      $ 538 "Direction: Base Z+"
      global move_thread_flag_538=0
      thread move_thread_538():
        enter_critical
        move_thread_flag_538 = 1
        local towardsPos=calculate_point_to_move_towards(p[0.0,0.0,0.0,0.0,0.0,0.0], [0.0,0.0,1.0], 0.06)
        movel(towardsPos, a=0.035, v=0.03)
        move_thread_flag_538 = 2
        exit_critical
      end
      move_thread_flag_538 = 0
      move_thread_han_538 = run move_thread_538()
      while (True):
        sleep(1.0E-10)
        if (move_thread_flag_538 > 1):
          join move_thread_han_538
          $ 539 "Until (distance)"
          break
        end
        sync()
      end
      $ 540 "Set CO[1]=Apagar"
      set_configurable_digital_out(1, False)
      $ 541 "barreno_actual≔barreno_actual+1"
      global barreno_actual=barreno_actual+1
      $ 542 "Call Quitar_broca"
      Quitar_broca()
      $ 543 "Call Poner_broca"
      Poner_broca()
    end
    $ 544 "CD"
    $ 545 "'desbaste_inicial'"
    # 'desbaste_inicial'
    $ 546 "bajada_broca≔p[0,0,-0.012,0,0,0]"
    global bajada_broca=p[0,0,-0.012,0,0,0]
    $ 547 "barrenos_menos1≔8"
    global barrenos_menos1=8
    $ 548 "barreno_actual≔0"
    global barreno_actual=0
    $ 549 "Loop barreno_actual≤barrenos_menos1"
    while (barreno_actual <= barrenos_menos1):
      $ 550 "Perforacion"
      $ 551 "MoveL"
      $ 552 "internos≔interpolate_pose(Linea1_C, Linea1_D, barreno_actual/barrenos_menos1)"
      global internos= interpolate_pose (Linea1_C_p, Linea1_D_p, barreno_actual/barrenos_menos1)
      $ 553 "internos" "breakAfter"
      movel(internos, a=0.5, v=0.1)
      $ 554 "'desbaste_inicial'"
      # 'desbaste_inicial'
      $ 555 "bajada_broca≔p[0,0,-0.024,0,0,0]"
      global bajada_broca=p[0,0,-0.024,0,0,0]
      $ 556 "bajada≔p[0,0,0.024,0,0,0]"
      global bajada=p[0,0,0.024,0,0,0]
      $ 557 "Direction: Base Z-"
      global move_thread_flag_557=0
      thread move_thread_557():
        enter_critical
        move_thread_flag_557 = 1
        local towardsPos=calculate_point_to_move_towards(p[0.0,0.0,0.0,0.0,0.0,0.0], [0.0,0.0,-1.0], 0.072)
        movel(towardsPos, a=0.035, v=0.03)
        move_thread_flag_557 = 2
        exit_critical
      end
      move_thread_flag_557 = 0
      move_thread_han_557 = run move_thread_557()
      while (True):
        sleep(1.0E-10)
        if (move_thread_flag_557 > 1):
          join move_thread_han_557
          $ 558 "Until (distance)"
          break
        end
        sync()
      end
      $ 559 "Popup: punto contacto alanzdo"
      popup("punto contacto alanzdo", "Mensaje", False, False, blocking=True)
      $ 560 "Direction: Base Z+"
      global move_thread_flag_560=0
      thread move_thread_560():
        enter_critical
        move_thread_flag_560 = 1
        local towardsPos=calculate_point_to_move_towards(p[0.0,0.0,0.0,0.0,0.0,0.0], [0.0,0.0,1.0], 0.002)
        movel(towardsPos, a=0.005, v=0.003)
        move_thread_flag_560 = 2
        exit_critical
      end
      move_thread_flag_560 = 0
      move_thread_han_560 = run move_thread_560()
      while (True):
        sleep(1.0E-10)
        if (move_thread_flag_560 > 1):
          join move_thread_han_560
          $ 561 "Until (distance)"
          break
        end
        sync()
      end
      $ 562 "Wait: 0.3"
      sleep(0.3)
      $ 563 "Set CO[1]=Encender"
      set_configurable_digital_out(1, True)
      $ 564 "Wait: 0.3"
      sleep(0.3)
      $ 565 "Loop 1 times"
      Loop_85 = 0
      while (Loop_85 < 1):
        $ 566 "bajar≔pose_add(get_actual_tcp_pose(), bajada_broca)"
        global bajar= pose_add ( get_actual_tcp_pose (), bajada_broca)
        $ 567 "bajar" "breakAfter"
        movel(bajar, a=0.005, v=0.001)
        $ 568 "subir≔pose_sub(get_actual_tcp_pose(), bajada_broca)"
        global subir= pose_sub ( get_actual_tcp_pose (), bajada_broca)
        $ 569 "subir" "breakAfter"
        movel(subir, a=0.01, v=0.005)
        $ 570 "bajada_broca≔pose_sub(bajada_broca, bajada)"
        global bajada_broca= pose_sub (bajada_broca, bajada)
        Loop_85 = Loop_85 + 1
      end
      $ 571 "Direction: Base Z+"
      global move_thread_flag_571=0
      thread move_thread_571():
        enter_critical
        move_thread_flag_571 = 1
        local towardsPos=calculate_point_to_move_towards(p[0.0,0.0,0.0,0.0,0.0,0.0], [0.0,0.0,1.0], 0.06)
        movel(towardsPos, a=0.035, v=0.03)
        move_thread_flag_571 = 2
        exit_critical
      end
      move_thread_flag_571 = 0
      move_thread_han_571 = run move_thread_571()
      while (True):
        sleep(1.0E-10)
        if (move_thread_flag_571 > 1):
          join move_thread_han_571
          $ 572 "Until (distance)"
          break
        end
        sync()
      end
      $ 573 "Set CO[1]=Apagar"
      set_configurable_digital_out(1, False)
      $ 574 "barreno_actual≔barreno_actual+1"
      global barreno_actual=barreno_actual+1
      $ 575 "Call Quitar_broca"
      Quitar_broca()
      $ 576 "Call Poner_broca"
      Poner_broca()
    end
    $ 577 "EF"
    $ 578 "'desbaste_inicial'"
    # 'desbaste_inicial'
    $ 579 "bajada_broca≔p[0,0,-0.012,0,0,0]"
    global bajada_broca=p[0,0,-0.012,0,0,0]
    $ 580 "barrenos_menos1≔8"
    global barrenos_menos1=8
    $ 581 "barreno_actual≔0"
    global barreno_actual=0
    $ 582 "Loop barreno_actual≤barrenos_menos1"
    while (barreno_actual <= barrenos_menos1):
      $ 583 "Perforacion"
      $ 584 "MoveL"
      $ 585 "internos≔interpolate_pose(Linea1_E, Linea1_F, barreno_actual/barrenos_menos1)"
      global internos= interpolate_pose (Linea1_E_p, Linea1_F_p, barreno_actual/barrenos_menos1)
      $ 586 "internos" "breakAfter"
      movel(internos, a=0.5, v=0.1)
      $ 587 "'desbaste_inicial'"
      # 'desbaste_inicial'
      $ 588 "bajada_broca≔p[0,0,-0.024,0,0,0]"
      global bajada_broca=p[0,0,-0.024,0,0,0]
      $ 589 "bajada≔p[0,0,0.024,0,0,0]"
      global bajada=p[0,0,0.024,0,0,0]
      $ 590 "Direction: Base Z-"
      global move_thread_flag_590=0
      thread move_thread_590():
        enter_critical
        move_thread_flag_590 = 1
        local towardsPos=calculate_point_to_move_towards(p[0.0,0.0,0.0,0.0,0.0,0.0], [0.0,0.0,-1.0], 0.072)
        movel(towardsPos, a=0.035, v=0.03)
        move_thread_flag_590 = 2
        exit_critical
      end
      move_thread_flag_590 = 0
      move_thread_han_590 = run move_thread_590()
      while (True):
        sleep(1.0E-10)
        if (move_thread_flag_590 > 1):
          join move_thread_han_590
          $ 591 "Until (distance)"
          break
        end
        sync()
      end
      $ 592 "Popup: punto contacto alanzdo"
      popup("punto contacto alanzdo", "Mensaje", False, False, blocking=True)
      $ 593 "Direction: Base Z+"
      global move_thread_flag_593=0
      thread move_thread_593():
        enter_critical
        move_thread_flag_593 = 1
        local towardsPos=calculate_point_to_move_towards(p[0.0,0.0,0.0,0.0,0.0,0.0], [0.0,0.0,1.0], 0.002)
        movel(towardsPos, a=0.005, v=0.003)
        move_thread_flag_593 = 2
        exit_critical
      end
      move_thread_flag_593 = 0
      move_thread_han_593 = run move_thread_593()
      while (True):
        sleep(1.0E-10)
        if (move_thread_flag_593 > 1):
          join move_thread_han_593
          $ 594 "Until (distance)"
          break
        end
        sync()
      end
      $ 595 "Wait: 0.3"
      sleep(0.3)
      $ 596 "Set CO[1]=Encender"
      set_configurable_digital_out(1, True)
      $ 597 "Wait: 0.3"
      sleep(0.3)
      $ 598 "Loop 1 times"
      Loop_87 = 0
      while (Loop_87 < 1):
        $ 599 "bajar≔pose_add(get_actual_tcp_pose(), bajada_broca)"
        global bajar= pose_add ( get_actual_tcp_pose (), bajada_broca)
        $ 600 "bajar" "breakAfter"
        movel(bajar, a=0.005, v=0.001)
        $ 601 "subir≔pose_sub(get_actual_tcp_pose(), bajada_broca)"
        global subir= pose_sub ( get_actual_tcp_pose (), bajada_broca)
        $ 602 "subir" "breakAfter"
        movel(subir, a=0.01, v=0.005)
        $ 603 "bajada_broca≔pose_sub(bajada_broca, bajada)"
        global bajada_broca= pose_sub (bajada_broca, bajada)
        Loop_87 = Loop_87 + 1
      end
      $ 604 "Direction: Base Z+"
      global move_thread_flag_604=0
      thread move_thread_604():
        enter_critical
        move_thread_flag_604 = 1
        local towardsPos=calculate_point_to_move_towards(p[0.0,0.0,0.0,0.0,0.0,0.0], [0.0,0.0,1.0], 0.06)
        movel(towardsPos, a=0.035, v=0.03)
        move_thread_flag_604 = 2
        exit_critical
      end
      move_thread_flag_604 = 0
      move_thread_han_604 = run move_thread_604()
      while (True):
        sleep(1.0E-10)
        if (move_thread_flag_604 > 1):
          join move_thread_han_604
          $ 605 "Until (distance)"
          break
        end
        sync()
      end
      $ 606 "Set CO[1]=Apagar"
      set_configurable_digital_out(1, False)
      $ 607 "barreno_actual≔barreno_actual+1"
      global barreno_actual=barreno_actual+1
      $ 608 "Call Quitar_broca"
      Quitar_broca()
      $ 609 "Call Poner_broca"
      Poner_broca()
    end
    $ 610 "Popup: Linea1 con full Terminada!"
    popup("Linea1 con full Terminada!", "Mensaje", False, False, blocking=True)
    $ 611 "Linea2"
    $ 612 "Marcar_puntos"
    $ 613 "MoveL"
    $ 614 "Home2" "breakAfter"
    movel(Home2_p, a=0.5, v=0.1)
    $ 623 "Linea2_A" "breakAfter"
    movel(Linea2_A_p, a=0.5, v=0.1)
    $ 624 "Linea2_B" "breakAfter"
    movel(Linea2_B_p, a=0.5, v=0.1)
    $ 625 "Linea2_C" "breakAfter"
    movel(Linea2_C_p, a=0.5, v=0.1)
    $ 626 "Linea2_D" "breakAfter"
    movel(Linea2_D_p, a=0.5, v=0.1)
    $ 627 "Linea2_E" "breakAfter"
    movel(Linea2_E_p, a=0.5, v=0.1)
    $ 628 "Linea2_F" "breakAfter"
    movel(Linea2_F_p, a=0.5, v=0.1)
    $ 629 "AB"
    $ 630 "'desbaste_inicial'"
    # 'desbaste_inicial'
    $ 631 "bajada_broca≔p[0,0,-0.012,0,0,0]"
    global bajada_broca=p[0,0,-0.012,0,0,0]
    $ 632 "barrenos_menos1≔8"
    global barrenos_menos1=8
    $ 633 "barreno_actual≔1"
    global barreno_actual=1
    $ 634 "Loop barreno_actual≤barrenos_menos1"
    while (barreno_actual <= barrenos_menos1):
      $ 635 "Perforacion"
      $ 636 "MoveL"
      $ 637 "internos≔interpolate_pose(Linea2_A, Linea2_B, barreno_actual/barrenos_menos1)"
      global internos= interpolate_pose (Linea2_A_p, Linea2_B_p, barreno_actual/barrenos_menos1)
      $ 638 "internos" "breakAfter"
      movel(internos, a=0.5, v=0.1)
      $ 639 "'desbaste_inicial'"
      # 'desbaste_inicial'
      $ 640 "bajada_broca≔p[0,0,-0.024,0,0,0]"
      global bajada_broca=p[0,0,-0.024,0,0,0]
      $ 641 "bajada≔p[0,0,0.024,0,0,0]"
      global bajada=p[0,0,0.024,0,0,0]
      $ 642 "Direction: Base Z-"
      global move_thread_flag_642=0
      thread move_thread_642():
        enter_critical
        move_thread_flag_642 = 1
        local towardsPos=calculate_point_to_move_towards(p[0.0,0.0,0.0,0.0,0.0,0.0], [0.0,0.0,-1.0], 0.076)
        movel(towardsPos, a=0.035, v=0.03)
        move_thread_flag_642 = 2
        exit_critical
      end
      move_thread_flag_642 = 0
      move_thread_han_642 = run move_thread_642()
      while (True):
        sleep(1.0E-10)
        if (move_thread_flag_642 > 1):
          join move_thread_han_642
          $ 643 "Until (distance)"
          break
        end
        sync()
      end
      $ 644 "Popup: punto contacto alanzdo"
      popup("punto contacto alanzdo", "Mensaje", False, False, blocking=True)
      $ 645 "Direction: Base Z+"
      global move_thread_flag_645=0
      thread move_thread_645():
        enter_critical
        move_thread_flag_645 = 1
        local towardsPos=calculate_point_to_move_towards(p[0.0,0.0,0.0,0.0,0.0,0.0], [0.0,0.0,1.0], 0.002)
        movel(towardsPos, a=0.005, v=0.003)
        move_thread_flag_645 = 2
        exit_critical
      end
      move_thread_flag_645 = 0
      move_thread_han_645 = run move_thread_645()
      while (True):
        sleep(1.0E-10)
        if (move_thread_flag_645 > 1):
          join move_thread_han_645
          $ 646 "Until (distance)"
          break
        end
        sync()
      end
      $ 647 "Wait: 0.3"
      sleep(0.3)
      $ 648 "Set CO[1]=Encender"
      set_configurable_digital_out(1, True)
      $ 649 "Wait: 0.3"
      sleep(0.3)
      $ 650 "Loop 1 times"
      Loop_90 = 0
      while (Loop_90 < 1):
        $ 651 "bajar≔pose_add(get_actual_tcp_pose(), bajada_broca)"
        global bajar= pose_add ( get_actual_tcp_pose (), bajada_broca)
        $ 652 "bajar" "breakAfter"
        movel(bajar, a=0.005, v=0.001)
        $ 653 "subir≔pose_sub(get_actual_tcp_pose(), bajada_broca)"
        global subir= pose_sub ( get_actual_tcp_pose (), bajada_broca)
        $ 654 "subir" "breakAfter"
        movel(subir, a=0.01, v=0.005)
        $ 655 "bajada_broca≔pose_sub(bajada_broca, bajada)"
        global bajada_broca= pose_sub (bajada_broca, bajada)
        Loop_90 = Loop_90 + 1
      end
      $ 656 "Direction: Base Z+"
      global move_thread_flag_656=0
      thread move_thread_656():
        enter_critical
        move_thread_flag_656 = 1
        local towardsPos=calculate_point_to_move_towards(p[0.0,0.0,0.0,0.0,0.0,0.0], [0.0,0.0,1.0], 0.06)
        movel(towardsPos, a=0.035, v=0.03)
        move_thread_flag_656 = 2
        exit_critical
      end
      move_thread_flag_656 = 0
      move_thread_han_656 = run move_thread_656()
      while (True):
        sleep(1.0E-10)
        if (move_thread_flag_656 > 1):
          join move_thread_han_656
          $ 657 "Until (distance)"
          break
        end
        sync()
      end
      $ 658 "Set CO[1]=Apagar"
      set_configurable_digital_out(1, False)
      $ 659 "barreno_actual≔barreno_actual+1"
      global barreno_actual=barreno_actual+1
      $ 660 "Call Quitar_broca"
      Quitar_broca()
      $ 661 "Call Poner_broca"
      Poner_broca()
    end
    $ 662 "CD"
    $ 663 "'desbaste_inicial'"
    # 'desbaste_inicial'
    $ 664 "bajada_broca≔p[0,0,-0.012,0,0,0]"
    global bajada_broca=p[0,0,-0.012,0,0,0]
    $ 665 "barrenos_menos1≔8"
    global barrenos_menos1=8
    $ 666 "barreno_actual≔0"
    global barreno_actual=0
    $ 667 "Loop barreno_actual≤barrenos_menos1"
    while (barreno_actual <= barrenos_menos1):
      $ 668 "Perforacion"
      $ 669 "MoveL"
      $ 670 "internos≔interpolate_pose(Linea2_C, Linea2_D, barreno_actual/barrenos_menos1)"
      global internos= interpolate_pose (Linea2_C_p, Linea2_D_p, barreno_actual/barrenos_menos1)
      $ 671 "internos" "breakAfter"
      movel(internos, a=0.5, v=0.1)
      $ 672 "'desbaste_inicial'"
      # 'desbaste_inicial'
      $ 673 "bajada_broca≔p[0,0,-0.024,0,0,0]"
      global bajada_broca=p[0,0,-0.024,0,0,0]
      $ 674 "bajada≔p[0,0,0.024,0,0,0]"
      global bajada=p[0,0,0.024,0,0,0]
      $ 675 "Direction: Base Z-"
      global move_thread_flag_675=0
      thread move_thread_675():
        enter_critical
        move_thread_flag_675 = 1
        local towardsPos=calculate_point_to_move_towards(p[0.0,0.0,0.0,0.0,0.0,0.0], [0.0,0.0,-1.0], 0.076)
        movel(towardsPos, a=0.035, v=0.03)
        move_thread_flag_675 = 2
        exit_critical
      end
      move_thread_flag_675 = 0
      move_thread_han_675 = run move_thread_675()
      while (True):
        sleep(1.0E-10)
        if (move_thread_flag_675 > 1):
          join move_thread_han_675
          $ 676 "Until (distance)"
          break
        end
        sync()
      end
      $ 677 "Popup: punto contacto alanzdo"
      popup("punto contacto alanzdo", "Mensaje", False, False, blocking=True)
      $ 678 "Direction: Base Z+"
      global move_thread_flag_678=0
      thread move_thread_678():
        enter_critical
        move_thread_flag_678 = 1
        local towardsPos=calculate_point_to_move_towards(p[0.0,0.0,0.0,0.0,0.0,0.0], [0.0,0.0,1.0], 0.002)
        movel(towardsPos, a=0.005, v=0.003)
        move_thread_flag_678 = 2
        exit_critical
      end
      move_thread_flag_678 = 0
      move_thread_han_678 = run move_thread_678()
      while (True):
        sleep(1.0E-10)
        if (move_thread_flag_678 > 1):
          join move_thread_han_678
          $ 679 "Until (distance)"
          break
        end
        sync()
      end
      $ 680 "Wait: 0.3"
      sleep(0.3)
      $ 681 "Set CO[1]=Encender"
      set_configurable_digital_out(1, True)
      $ 682 "Wait: 0.3"
      sleep(0.3)
      $ 683 "Loop 1 times"
      Loop_92 = 0
      while (Loop_92 < 1):
        $ 684 "bajar≔pose_add(get_actual_tcp_pose(), bajada_broca)"
        global bajar= pose_add ( get_actual_tcp_pose (), bajada_broca)
        $ 685 "bajar" "breakAfter"
        movel(bajar, a=0.005, v=0.001)
        $ 686 "subir≔pose_sub(get_actual_tcp_pose(), bajada_broca)"
        global subir= pose_sub ( get_actual_tcp_pose (), bajada_broca)
        $ 687 "subir" "breakAfter"
        movel(subir, a=0.01, v=0.005)
        $ 688 "bajada_broca≔pose_sub(bajada_broca, bajada)"
        global bajada_broca= pose_sub (bajada_broca, bajada)
        Loop_92 = Loop_92 + 1
      end
      $ 689 "Direction: Base Z+"
      global move_thread_flag_689=0
      thread move_thread_689():
        enter_critical
        move_thread_flag_689 = 1
        local towardsPos=calculate_point_to_move_towards(p[0.0,0.0,0.0,0.0,0.0,0.0], [0.0,0.0,1.0], 0.06)
        movel(towardsPos, a=0.035, v=0.03)
        move_thread_flag_689 = 2
        exit_critical
      end
      move_thread_flag_689 = 0
      move_thread_han_689 = run move_thread_689()
      while (True):
        sleep(1.0E-10)
        if (move_thread_flag_689 > 1):
          join move_thread_han_689
          $ 690 "Until (distance)"
          break
        end
        sync()
      end
      $ 691 "Set CO[1]=Apagar"
      set_configurable_digital_out(1, False)
      $ 692 "barreno_actual≔barreno_actual+1"
      global barreno_actual=barreno_actual+1
      $ 693 "Call Quitar_broca"
      Quitar_broca()
      $ 694 "Call Poner_broca"
      Poner_broca()
    end
    $ 695 "EF"
    $ 696 "'desbaste_inicial'"
    # 'desbaste_inicial'
    $ 697 "bajada_broca≔p[0,0,-0.012,0,0,0]"
    global bajada_broca=p[0,0,-0.012,0,0,0]
    $ 698 "barrenos_menos1≔8"
    global barrenos_menos1=8
    $ 699 "barreno_actual≔0"
    global barreno_actual=0
    $ 700 "Loop barreno_actual≤barrenos_menos1"
    while (barreno_actual <= barrenos_menos1):
      $ 701 "Perforacion"
      $ 702 "MoveL"
      $ 703 "internos≔interpolate_pose(Linea2_E, Linea2_F, barreno_actual/barrenos_menos1)"
      global internos= interpolate_pose (Linea2_E_p, Linea2_F_p, barreno_actual/barrenos_menos1)
      $ 704 "internos" "breakAfter"
      movel(internos, a=0.5, v=0.1)
      $ 705 "'desbaste_inicial'"
      # 'desbaste_inicial'
      $ 706 "bajada_broca≔p[0,0,-0.024,0,0,0]"
      global bajada_broca=p[0,0,-0.024,0,0,0]
      $ 707 "bajada≔p[0,0,0.024,0,0,0]"
      global bajada=p[0,0,0.024,0,0,0]
      $ 708 "Direction: Base Z-"
      global move_thread_flag_708=0
      thread move_thread_708():
        enter_critical
        move_thread_flag_708 = 1
        local towardsPos=calculate_point_to_move_towards(p[0.0,0.0,0.0,0.0,0.0,0.0], [0.0,0.0,-1.0], 0.076)
        movel(towardsPos, a=0.035, v=0.03)
        move_thread_flag_708 = 2
        exit_critical
      end
      move_thread_flag_708 = 0
      move_thread_han_708 = run move_thread_708()
      while (True):
        sleep(1.0E-10)
        if (move_thread_flag_708 > 1):
          join move_thread_han_708
          $ 709 "Until (distance)"
          break
        end
        sync()
      end
      $ 710 "Popup: punto contacto alanzdo"
      popup("punto contacto alanzdo", "Mensaje", False, False, blocking=True)
      $ 711 "Direction: Base Z+"
      global move_thread_flag_711=0
      thread move_thread_711():
        enter_critical
        move_thread_flag_711 = 1
        local towardsPos=calculate_point_to_move_towards(p[0.0,0.0,0.0,0.0,0.0,0.0], [0.0,0.0,1.0], 0.002)
        movel(towardsPos, a=0.015, v=0.015)
        move_thread_flag_711 = 2
        exit_critical
      end
      move_thread_flag_711 = 0
      move_thread_han_711 = run move_thread_711()
      while (True):
        sleep(1.0E-10)
        if (move_thread_flag_711 > 1):
          join move_thread_han_711
          $ 712 "Until (distance)"
          break
        end
        sync()
      end
      $ 713 "Wait: 0.3"
      sleep(0.3)
      $ 714 "Set CO[1]=Encender"
      set_configurable_digital_out(1, True)
      $ 715 "Wait: 0.3"
      sleep(0.3)
      $ 716 "Loop 1 times"
      Loop_94 = 0
      while (Loop_94 < 1):
        $ 717 "bajar≔pose_add(get_actual_tcp_pose(), bajada_broca)"
        global bajar= pose_add ( get_actual_tcp_pose (), bajada_broca)
        $ 718 "bajar" "breakAfter"
        movel(bajar, a=0.005, v=0.001)
        $ 719 "subir≔pose_sub(get_actual_tcp_pose(), bajada_broca)"
        global subir= pose_sub ( get_actual_tcp_pose (), bajada_broca)
        $ 720 "subir" "breakAfter"
        movel(subir, a=0.01, v=0.005)
        $ 721 "bajada_broca≔pose_sub(bajada_broca, bajada)"
        global bajada_broca= pose_sub (bajada_broca, bajada)
        Loop_94 = Loop_94 + 1
      end
      $ 722 "Direction: Base Z+"
      global move_thread_flag_722=0
      thread move_thread_722():
        enter_critical
        move_thread_flag_722 = 1
        local towardsPos=calculate_point_to_move_towards(p[0.0,0.0,0.0,0.0,0.0,0.0], [0.0,0.0,1.0], 0.06)
        movel(towardsPos, a=0.035, v=0.03)
        move_thread_flag_722 = 2
        exit_critical
      end
      move_thread_flag_722 = 0
      move_thread_han_722 = run move_thread_722()
      while (True):
        sleep(1.0E-10)
        if (move_thread_flag_722 > 1):
          join move_thread_han_722
          $ 723 "Until (distance)"
          break
        end
        sync()
      end
      $ 724 "Set CO[1]=Apagar"
      set_configurable_digital_out(1, False)
      $ 725 "barreno_actual≔barreno_actual+1"
      global barreno_actual=barreno_actual+1
      $ 726 "If barreno_actual>barrenos_menos1"
      if (barreno_actual>barrenos_menos1):
        $ 727 "cambiar_broca≔ True "
        global cambiar_broca=  True
      end
      $ 728 "Call Quitar_broca"
      Quitar_broca()
      $ 729 "Call Poner_broca"
      Poner_broca()
    end
    $ 730 "Popup: Linea2 con full Terminada!"
    popup("Linea2 con full Terminada!", "Mensaje", False, False, blocking=True)
    $ 731 "600"
    $ 1243 "Broca_1"
    $ 1244 "Linea7"
    $ 1245 "Marcar_puntos"
    $ 1246 "MoveL"
    $ 1247 "Home2" "breakAfter"
    movel(Home2_p, a=0.5, v=0.1)
    $ 1248 "Linea7_A" "breakAfter"
    movel(Linea7_A_p, a=0.5, v=0.1)
    $ 1249 "bajada_comprobacion"
    $ 1250 "Direction: Base Z-"
    global move_thread_flag_1250=0
    thread move_thread_1250():
      enter_critical
      move_thread_flag_1250 = 1
      local towardsPos=calculate_point_to_move_towards(p[0.0,0.0,0.0,0.0,0.0,0.0], [0.0,0.0,-1.0], 0.071)
      movel(towardsPos, a=0.15, v=0.1)
      move_thread_flag_1250 = 2
      exit_critical
    end
    move_thread_flag_1250 = 0
    move_thread_han_1250 = run move_thread_1250()
    while (True):
      sleep(1.0E-10)
      if (move_thread_flag_1250 > 1):
        join move_thread_han_1250
        $ 1251 "Until (distance)"
        break
      end
      sync()
    end
    $ 1252 "Direction: Base Z-"
    global move_thread_flag_1252=0
    thread move_thread_1252():
      enter_critical
      move_thread_flag_1252 = 1
      local towardsPos=calculate_point_to_move_towards(p[0.0,0.0,0.0,0.0,0.0,0.0], [0.0,0.0,-1.0], 1000.0)
      movel(towardsPos, a=0.007, v=0.007)
      move_thread_flag_1252 = 2
      exit_critical
    end
    move_thread_flag_1252 = 0
    move_thread_han_1252 = run move_thread_1252()
    while (True):
      local targetTcpDirection=get_target_tcp_speed()
      local stepsToRetract=tool_contact(direction=targetTcpDirection)
      if (stepsToRetract > 0):
        kill move_thread_han_1252
        stopl(0.02)
        local backTrackMovement=get_actual_joint_positions_history(stepsToRetract)
        local contactPose=get_forward_kin(backTrackMovement)
        local posDir=[targetTcpDirection[0],targetTcpDirection[1],targetTcpDirection[2]]
        local retractTo=contactPose
        if (norm(posDir) > 1e-6):
          local normalizedPosDir=normalize(posDir)
          local additionalRetraction=p[normalizedPosDir[0] * 0.0, normalizedPosDir[1] * 0.0, normalizedPosDir[2] * 0.0, 0, 0, 0]
          retractTo = pose_sub(contactPose, additionalRetraction)
        end
        movel(retractTo, a=0.02, v=0.1)
        $ 1253 "Until (tool_contact_detection)"
        break
      end
      sync()
    end
    $ 1254 "Direction: Base Z+"
    global move_thread_flag_1254=0
    thread move_thread_1254():
      enter_critical
      move_thread_flag_1254 = 1
      local towardsPos=calculate_point_to_move_towards(p[0.0,0.0,0.0,0.0,0.0,0.0], [0.0,0.0,1.0], 0.08)
      movel(towardsPos, a=0.15, v=0.1)
      move_thread_flag_1254 = 2
      exit_critical
    end
    move_thread_flag_1254 = 0
    move_thread_han_1254 = run move_thread_1254()
    while (True):
      sleep(1.0E-10)
      if (move_thread_flag_1254 > 1):
        join move_thread_han_1254
        $ 1255 "Until (distance)"
        break
      end
      sync()
    end
    $ 1256 "Linea7_B" "breakAfter"
    movel(Linea7_B_p, a=0.5, v=0.1)
    $ 1257 "bajada_comprobacion"
    $ 1258 "Direction: Base Z-"
    global move_thread_flag_1258=0
    thread move_thread_1258():
      enter_critical
      move_thread_flag_1258 = 1
      local towardsPos=calculate_point_to_move_towards(p[0.0,0.0,0.0,0.0,0.0,0.0], [0.0,0.0,-1.0], 0.071)
      movel(towardsPos, a=0.15, v=0.1)
      move_thread_flag_1258 = 2
      exit_critical
    end
    move_thread_flag_1258 = 0
    move_thread_han_1258 = run move_thread_1258()
    while (True):
      sleep(1.0E-10)
      if (move_thread_flag_1258 > 1):
        join move_thread_han_1258
        $ 1259 "Until (distance)"
        break
      end
      sync()
    end
    $ 1260 "Direction: Base Z-"
    global move_thread_flag_1260=0
    thread move_thread_1260():
      enter_critical
      move_thread_flag_1260 = 1
      local towardsPos=calculate_point_to_move_towards(p[0.0,0.0,0.0,0.0,0.0,0.0], [0.0,0.0,-1.0], 1000.0)
      movel(towardsPos, a=0.007, v=0.007)
      move_thread_flag_1260 = 2
      exit_critical
    end
    move_thread_flag_1260 = 0
    move_thread_han_1260 = run move_thread_1260()
    while (True):
      local targetTcpDirection=get_target_tcp_speed()
      local stepsToRetract=tool_contact(direction=targetTcpDirection)
      if (stepsToRetract > 0):
        kill move_thread_han_1260
        stopl(0.02)
        local backTrackMovement=get_actual_joint_positions_history(stepsToRetract)
        local contactPose=get_forward_kin(backTrackMovement)
        local posDir=[targetTcpDirection[0],targetTcpDirection[1],targetTcpDirection[2]]
        local retractTo=contactPose
        if (norm(posDir) > 1e-6):
          local normalizedPosDir=normalize(posDir)
          local additionalRetraction=p[normalizedPosDir[0] * 0.0, normalizedPosDir[1] * 0.0, normalizedPosDir[2] * 0.0, 0, 0, 0]
          retractTo = pose_sub(contactPose, additionalRetraction)
        end
        movel(retractTo, a=0.02, v=0.1)
        $ 1261 "Until (tool_contact_detection)"
        break
      end
      sync()
    end
    $ 1262 "Direction: Base Z+"
    global move_thread_flag_1262=0
    thread move_thread_1262():
      enter_critical
      move_thread_flag_1262 = 1
      local towardsPos=calculate_point_to_move_towards(p[0.0,0.0,0.0,0.0,0.0,0.0], [0.0,0.0,1.0], 0.08)
      movel(towardsPos, a=0.15, v=0.1)
      move_thread_flag_1262 = 2
      exit_critical
    end
    move_thread_flag_1262 = 0
    move_thread_han_1262 = run move_thread_1262()
    while (True):
      sleep(1.0E-10)
      if (move_thread_flag_1262 > 1):
        join move_thread_han_1262
        $ 1263 "Until (distance)"
        break
      end
      sync()
    end
    $ 1264 "AB"
    $ 1265 "'desbaste_inicial'"
    # 'desbaste_inicial'
    $ 1266 "bajada_broca≔p[0,0,-0.008,0,0,0]"
    global bajada_broca=p[0,0,-0.008,0,0,0]
    $ 1267 "barrenos_menos1≔2"
    global barrenos_menos1=2
    $ 1268 "barreno_actual≔0"
    global barreno_actual=0
    $ 1269 "Loop barreno_actual≤barrenos_menos1"
    while (barreno_actual <= barrenos_menos1):
      $ 1270 "Perforacion"
      $ 1271 "MoveL"
      $ 1272 "internos≔interpolate_pose(Linea7_A, Linea7_B, barreno_actual/barrenos_menos1)"
      global internos= interpolate_pose (Linea7_A_p, Linea7_B_p, barreno_actual/barrenos_menos1)
      $ 1273 "internos" "breakAfter"
      movel(internos, a=0.5, v=0.1)
      $ 1274 "'desbaste_inicial'"
      # 'desbaste_inicial'
      $ 1275 "bajada_broca≔p[0,0,-0.024,0,0,0]"
      global bajada_broca=p[0,0,-0.024,0,0,0]
      $ 1276 "bajada≔p[0,0,0.024,0,0,0]"
      global bajada=p[0,0,0.024,0,0,0]
      $ 1277 "Direction: Base Z-"
      global move_thread_flag_1277=0
      thread move_thread_1277():
        enter_critical
        move_thread_flag_1277 = 1
        local towardsPos=calculate_point_to_move_towards(p[0.0,0.0,0.0,0.0,0.0,0.0], [0.0,0.0,-1.0], 0.071)
        movel(towardsPos, a=0.15, v=0.1)
        move_thread_flag_1277 = 2
        exit_critical
      end
      move_thread_flag_1277 = 0
      move_thread_han_1277 = run move_thread_1277()
      while (True):
        sleep(1.0E-10)
        if (move_thread_flag_1277 > 1):
          join move_thread_han_1277
          $ 1278 "Until (distance)"
          break
        end
        sync()
      end
      $ 1279 "Direction: Base Z-"
      global move_thread_flag_1279=0
      thread move_thread_1279():
        enter_critical
        move_thread_flag_1279 = 1
        local towardsPos=calculate_point_to_move_towards(p[0.0,0.0,0.0,0.0,0.0,0.0], [0.0,0.0,-1.0], 1000.0)
        movel(towardsPos, a=0.007, v=0.007)
        move_thread_flag_1279 = 2
        exit_critical
      end
      move_thread_flag_1279 = 0
      move_thread_han_1279 = run move_thread_1279()
      while (True):
        local targetTcpDirection=get_target_tcp_speed()
        local stepsToRetract=tool_contact(direction=targetTcpDirection)
        if (stepsToRetract > 0):
          kill move_thread_han_1279
          stopl(0.02)
          local backTrackMovement=get_actual_joint_positions_history(stepsToRetract)
          local contactPose=get_forward_kin(backTrackMovement)
          local posDir=[targetTcpDirection[0],targetTcpDirection[1],targetTcpDirection[2]]
          local retractTo=contactPose
          if (norm(posDir) > 1e-6):
            local normalizedPosDir=normalize(posDir)
            local additionalRetraction=p[normalizedPosDir[0] * 0.0, normalizedPosDir[1] * 0.0, normalizedPosDir[2] * 0.0, 0, 0, 0]
            retractTo = pose_sub(contactPose, additionalRetraction)
          end
          movel(retractTo, a=0.02, v=0.1)
          $ 1280 "Until (tool_contact_detection)"
          break
        end
        sync()
      end
      $ 1281 "Popup: punto contacto alanzdo"
      popup("punto contacto alanzdo", "Mensaje", False, False, blocking=True)
      $ 1282 "Direction: Base Z+"
      global move_thread_flag_1282=0
      thread move_thread_1282():
        enter_critical
        move_thread_flag_1282 = 1
        local towardsPos=calculate_point_to_move_towards(p[0.0,0.0,0.0,0.0,0.0,0.0], [0.0,0.0,1.0], 0.002)
        movel(towardsPos, a=0.005, v=0.003)
        move_thread_flag_1282 = 2
        exit_critical
      end
      move_thread_flag_1282 = 0
      move_thread_han_1282 = run move_thread_1282()
      while (True):
        sleep(1.0E-10)
        if (move_thread_flag_1282 > 1):
          join move_thread_han_1282
          $ 1283 "Until (distance)"
          break
        end
        sync()
      end
      $ 1284 "Wait: 0.3"
      sleep(0.3)
      $ 1285 "Set CO[1]=Encender"
      set_configurable_digital_out(1, True)
      $ 1286 "Wait: 0.3"
      sleep(0.3)
      $ 1287 "Loop 1 times"
      Loop_96 = 0
      while (Loop_96 < 1):
        $ 1288 "bajar≔pose_add(get_actual_tcp_pose(), bajada_broca)"
        global bajar= pose_add ( get_actual_tcp_pose (), bajada_broca)
        $ 1289 "bajar" "breakAfter"
        movel(bajar, a=0.01, v=0.01)
        $ 1290 "subir≔pose_sub(get_actual_tcp_pose(), bajada_broca)"
        global subir= pose_sub ( get_actual_tcp_pose (), bajada_broca)
        $ 1291 "subir" "breakAfter"
        movel(subir, a=0.015, v=0.015)
        $ 1292 "bajada_broca≔pose_sub(bajada_broca, bajada)"
        global bajada_broca= pose_sub (bajada_broca, bajada)
        Loop_96 = Loop_96 + 1
      end
      $ 1293 "Direction: Base Z+"
      global move_thread_flag_1293=0
      thread move_thread_1293():
        enter_critical
        move_thread_flag_1293 = 1
        local towardsPos=calculate_point_to_move_towards(p[0.0,0.0,0.0,0.0,0.0,0.0], [0.0,0.0,1.0], 0.08)
        movel(towardsPos, a=0.15, v=0.1)
        move_thread_flag_1293 = 2
        exit_critical
      end
      move_thread_flag_1293 = 0
      move_thread_han_1293 = run move_thread_1293()
      while (True):
        sleep(1.0E-10)
        if (move_thread_flag_1293 > 1):
          join move_thread_han_1293
          $ 1294 "Until (distance)"
          break
        end
        sync()
      end
      $ 1295 "Set CO[1]=Apagar"
      set_configurable_digital_out(1, False)
      $ 1296 "barreno_actual≔barreno_actual+1"
      global barreno_actual=barreno_actual+1
      $ 1297 "Call Quitar_broca"
      Quitar_broca()
      $ 1298 "Call Poner_broca"
      Poner_broca()
    end
    $ 1299 "Popup: Linea7 con chica Terminada!"
    popup("Linea7 con chica Terminada!", "Mensaje", False, False, blocking=True)
    $ 1300 "Linea8"
    $ 1301 "Marcar_puntos"
    $ 1302 "MoveL"
    $ 1303 "Linea8_A" "breakAfter"
    movel(Linea8_A_p, a=0.5, v=0.1)
    $ 1304 "bajada_comprobacion"
    $ 1305 "Direction: Base Z-"
    global move_thread_flag_1305=0
    thread move_thread_1305():
      enter_critical
      move_thread_flag_1305 = 1
      local towardsPos=calculate_point_to_move_towards(p[0.0,0.0,0.0,0.0,0.0,0.0], [0.0,0.0,-1.0], 0.071)
      movel(towardsPos, a=0.15, v=0.1)
      move_thread_flag_1305 = 2
      exit_critical
    end
    move_thread_flag_1305 = 0
    move_thread_han_1305 = run move_thread_1305()
    while (True):
      sleep(1.0E-10)
      if (move_thread_flag_1305 > 1):
        join move_thread_han_1305
        $ 1306 "Until (distance)"
        break
      end
      sync()
    end
    $ 1307 "Direction: Base Z-"
    global move_thread_flag_1307=0
    thread move_thread_1307():
      enter_critical
      move_thread_flag_1307 = 1
      local towardsPos=calculate_point_to_move_towards(p[0.0,0.0,0.0,0.0,0.0,0.0], [0.0,0.0,-1.0], 1000.0)
      movel(towardsPos, a=0.007, v=0.007)
      move_thread_flag_1307 = 2
      exit_critical
    end
    move_thread_flag_1307 = 0
    move_thread_han_1307 = run move_thread_1307()
    while (True):
      local targetTcpDirection=get_target_tcp_speed()
      local stepsToRetract=tool_contact(direction=targetTcpDirection)
      if (stepsToRetract > 0):
        kill move_thread_han_1307
        stopl(0.007)
        local backTrackMovement=get_actual_joint_positions_history(stepsToRetract)
        local contactPose=get_forward_kin(backTrackMovement)
        local posDir=[targetTcpDirection[0],targetTcpDirection[1],targetTcpDirection[2]]
        local retractTo=contactPose
        if (norm(posDir) > 1e-6):
          local normalizedPosDir=normalize(posDir)
          local additionalRetraction=p[normalizedPosDir[0] * 0.0, normalizedPosDir[1] * 0.0, normalizedPosDir[2] * 0.0, 0, 0, 0]
          retractTo = pose_sub(contactPose, additionalRetraction)
        end
        movel(retractTo, a=0.007, v=0.1)
        $ 1308 "Until (tool_contact_detection)"
        break
      end
      sync()
    end
    $ 1309 "Direction: Base Z+"
    global move_thread_flag_1309=0
    thread move_thread_1309():
      enter_critical
      move_thread_flag_1309 = 1
      local towardsPos=calculate_point_to_move_towards(p[0.0,0.0,0.0,0.0,0.0,0.0], [0.0,0.0,1.0], 0.08)
      movel(towardsPos, a=0.15, v=0.1)
      move_thread_flag_1309 = 2
      exit_critical
    end
    move_thread_flag_1309 = 0
    move_thread_han_1309 = run move_thread_1309()
    while (True):
      sleep(1.0E-10)
      if (move_thread_flag_1309 > 1):
        join move_thread_han_1309
        $ 1310 "Until (distance)"
        break
      end
      sync()
    end
    $ 1311 "Linea8_B" "breakAfter"
    movel(Linea8_B_p, a=0.5, v=0.1)
    $ 1312 "bajada_comprobacion"
    $ 1313 "Direction: Base Z-"
    global move_thread_flag_1313=0
    thread move_thread_1313():
      enter_critical
      move_thread_flag_1313 = 1
      local towardsPos=calculate_point_to_move_towards(p[0.0,0.0,0.0,0.0,0.0,0.0], [0.0,0.0,-1.0], 0.071)
      movel(towardsPos, a=0.15, v=0.1)
      move_thread_flag_1313 = 2
      exit_critical
    end
    move_thread_flag_1313 = 0
    move_thread_han_1313 = run move_thread_1313()
    while (True):
      sleep(1.0E-10)
      if (move_thread_flag_1313 > 1):
        join move_thread_han_1313
        $ 1314 "Until (distance)"
        break
      end
      sync()
    end
    $ 1315 "Direction: Base Z-"
    global move_thread_flag_1315=0
    thread move_thread_1315():
      enter_critical
      move_thread_flag_1315 = 1
      local towardsPos=calculate_point_to_move_towards(p[0.0,0.0,0.0,0.0,0.0,0.0], [0.0,0.0,-1.0], 1000.0)
      movel(towardsPos, a=0.007, v=0.007)
      move_thread_flag_1315 = 2
      exit_critical
    end
    move_thread_flag_1315 = 0
    move_thread_han_1315 = run move_thread_1315()
    while (True):
      local targetTcpDirection=get_target_tcp_speed()
      local stepsToRetract=tool_contact(direction=targetTcpDirection)
      if (stepsToRetract > 0):
        kill move_thread_han_1315
        stopl(0.007)
        local backTrackMovement=get_actual_joint_positions_history(stepsToRetract)
        local contactPose=get_forward_kin(backTrackMovement)
        local posDir=[targetTcpDirection[0],targetTcpDirection[1],targetTcpDirection[2]]
        local retractTo=contactPose
        if (norm(posDir) > 1e-6):
          local normalizedPosDir=normalize(posDir)
          local additionalRetraction=p[normalizedPosDir[0] * 0.0, normalizedPosDir[1] * 0.0, normalizedPosDir[2] * 0.0, 0, 0, 0]
          retractTo = pose_sub(contactPose, additionalRetraction)
        end
        movel(retractTo, a=0.007, v=0.1)
        $ 1316 "Until (tool_contact_detection)"
        break
      end
      sync()
    end
    $ 1317 "Direction: Base Z+"
    global move_thread_flag_1317=0
    thread move_thread_1317():
      enter_critical
      move_thread_flag_1317 = 1
      local towardsPos=calculate_point_to_move_towards(p[0.0,0.0,0.0,0.0,0.0,0.0], [0.0,0.0,1.0], 0.08)
      movel(towardsPos, a=0.15, v=0.1)
      move_thread_flag_1317 = 2
      exit_critical
    end
    move_thread_flag_1317 = 0
    move_thread_han_1317 = run move_thread_1317()
    while (True):
      sleep(1.0E-10)
      if (move_thread_flag_1317 > 1):
        join move_thread_han_1317
        $ 1318 "Until (distance)"
        break
      end
      sync()
    end
    $ 1319 "AB"
    $ 1320 "'desbaste_inicial'"
    # 'desbaste_inicial'
    $ 1321 "bajada_broca≔p[0,0,-0.008,0,0,0]"
    global bajada_broca=p[0,0,-0.008,0,0,0]
    $ 1322 "barrenos_menos1≔5"
    global barrenos_menos1=5
    $ 1323 "barreno_actual≔0"
    global barreno_actual=0
    $ 1324 "Loop barreno_actual≤barrenos_menos1"
    while (barreno_actual <= barrenos_menos1):
      $ 1325 "Perforacion"
      $ 1326 "MoveL"
      $ 1327 "internos≔interpolate_pose(Linea8_A, Linea8_B, barreno_actual/barrenos_menos1)"
      global internos= interpolate_pose (Linea8_A_p, Linea8_B_p, barreno_actual/barrenos_menos1)
      $ 1328 "internos" "breakAfter"
      movel(internos, a=0.5, v=0.1)
      $ 1329 "'desbaste_inicial'"
      # 'desbaste_inicial'
      $ 1330 "bajada_broca≔p[0,0,-0.024,0,0,0]"
      global bajada_broca=p[0,0,-0.024,0,0,0]
      $ 1331 "bajada≔p[0,0,0.0024,0,0,0]"
      global bajada=p[0,0,0.0024,0,0,0]
      $ 1332 "Direction: Base Z-"
      global move_thread_flag_1332=0
      thread move_thread_1332():
        enter_critical
        move_thread_flag_1332 = 1
        local towardsPos=calculate_point_to_move_towards(p[0.0,0.0,0.0,0.0,0.0,0.0], [0.0,0.0,-1.0], 0.071)
        movel(towardsPos, a=0.15, v=0.1)
        move_thread_flag_1332 = 2
        exit_critical
      end
      move_thread_flag_1332 = 0
      move_thread_han_1332 = run move_thread_1332()
      while (True):
        sleep(1.0E-10)
        if (move_thread_flag_1332 > 1):
          join move_thread_han_1332
          $ 1333 "Until (distance)"
          break
        end
        sync()
      end
      $ 1334 "Direction: Base Z-"
      global move_thread_flag_1334=0
      thread move_thread_1334():
        enter_critical
        move_thread_flag_1334 = 1
        local towardsPos=calculate_point_to_move_towards(p[0.0,0.0,0.0,0.0,0.0,0.0], [0.0,0.0,-1.0], 1000.0)
        movel(towardsPos, a=0.01, v=0.01)
        move_thread_flag_1334 = 2
        exit_critical
      end
      move_thread_flag_1334 = 0
      move_thread_han_1334 = run move_thread_1334()
      while (True):
        local targetTcpDirection=get_target_tcp_speed()
        local stepsToRetract=tool_contact(direction=targetTcpDirection)
        if (stepsToRetract > 0):
          kill move_thread_han_1334
          stopl(0.01)
          local backTrackMovement=get_actual_joint_positions_history(stepsToRetract)
          local contactPose=get_forward_kin(backTrackMovement)
          local posDir=[targetTcpDirection[0],targetTcpDirection[1],targetTcpDirection[2]]
          local retractTo=contactPose
          if (norm(posDir) > 1e-6):
            local normalizedPosDir=normalize(posDir)
            local additionalRetraction=p[normalizedPosDir[0] * 0.0, normalizedPosDir[1] * 0.0, normalizedPosDir[2] * 0.0, 0, 0, 0]
            retractTo = pose_sub(contactPose, additionalRetraction)
          end
          movel(retractTo, a=0.01, v=0.1)
          $ 1335 "Until (tool_contact_detection)"
          break
        end
        sync()
      end
      $ 1336 "Popup: punto contacto alanzdo"
      popup("punto contacto alanzdo", "Mensaje", False, False, blocking=True)
      $ 1337 "Direction: Base Z+"
      global move_thread_flag_1337=0
      thread move_thread_1337():
        enter_critical
        move_thread_flag_1337 = 1
        local towardsPos=calculate_point_to_move_towards(p[0.0,0.0,0.0,0.0,0.0,0.0], [0.0,0.0,1.0], 0.002)
        movel(towardsPos, a=0.005, v=0.003)
        move_thread_flag_1337 = 2
        exit_critical
      end
      move_thread_flag_1337 = 0
      move_thread_han_1337 = run move_thread_1337()
      while (True):
        sleep(1.0E-10)
        if (move_thread_flag_1337 > 1):
          join move_thread_han_1337
          $ 1338 "Until (distance)"
          break
        end
        sync()
      end
      $ 1339 "Wait: 0.3"
      sleep(0.3)
      $ 1340 "Set CO[1]=Encender"
      set_configurable_digital_out(1, True)
      $ 1341 "Wait: 0.3"
      sleep(0.3)
      $ 1342 "Loop 1 times"
      Loop_110 = 0
      while (Loop_110 < 1):
        $ 1343 "bajar≔pose_add(get_actual_tcp_pose(), bajada_broca)"
        global bajar= pose_add ( get_actual_tcp_pose (), bajada_broca)
        $ 1344 "bajar" "breakAfter"
        movel(bajar, a=0.01, v=0.01)
        $ 1345 "subir≔pose_sub(get_actual_tcp_pose(), bajada_broca)"
        global subir= pose_sub ( get_actual_tcp_pose (), bajada_broca)
        $ 1346 "subir" "breakAfter"
        movel(subir, a=0.015, v=0.015)
        $ 1347 "bajada_broca≔pose_sub(bajada_broca, bajada)"
        global bajada_broca= pose_sub (bajada_broca, bajada)
        Loop_110 = Loop_110 + 1
      end
      $ 1348 "Direction: Base Z+"
      global move_thread_flag_1348=0
      thread move_thread_1348():
        enter_critical
        move_thread_flag_1348 = 1
        local towardsPos=calculate_point_to_move_towards(p[0.0,0.0,0.0,0.0,0.0,0.0], [0.0,0.0,1.0], 0.08)
        movel(towardsPos, a=0.15, v=0.1)
        move_thread_flag_1348 = 2
        exit_critical
      end
      move_thread_flag_1348 = 0
      move_thread_han_1348 = run move_thread_1348()
      while (True):
        sleep(1.0E-10)
        if (move_thread_flag_1348 > 1):
          join move_thread_han_1348
          $ 1349 "Until (distance)"
          break
        end
        sync()
      end
      $ 1350 "Set CO[1]=Apagar"
      set_configurable_digital_out(1, False)
      $ 1351 "barreno_actual≔barreno_actual+1"
      global barreno_actual=barreno_actual+1
      $ 1352 "Call Quitar_broca"
      Quitar_broca()
      $ 1353 "Call Poner_broca"
      Poner_broca()
    end
    $ 1354 "Popup: Linea8 con chica Terminada!"
    popup("Linea8 con chica Terminada!", "Mensaje", False, False, blocking=True)
    $ 1355 "Linea9"
    $ 1356 "Marcar_puntos"
    $ 1357 "MoveL"
    $ 1358 "Linea9_A" "breakAfter"
    movel(Linea9_A_p, a=0.5, v=0.1)
    $ 1359 "bajada_comprobacion"
    $ 1360 "Direction: Base Z-"
    global move_thread_flag_1360=0
    thread move_thread_1360():
      enter_critical
      move_thread_flag_1360 = 1
      local towardsPos=calculate_point_to_move_towards(p[0.0,0.0,0.0,0.0,0.0,0.0], [0.0,0.0,-1.0], 0.071)
      movel(towardsPos, a=0.15, v=0.1)
      move_thread_flag_1360 = 2
      exit_critical
    end
    move_thread_flag_1360 = 0
    move_thread_han_1360 = run move_thread_1360()
    while (True):
      sleep(1.0E-10)
      if (move_thread_flag_1360 > 1):
        join move_thread_han_1360
        $ 1361 "Until (distance)"
        break
      end
      sync()
    end
    $ 1362 "Direction: Base Z-"
    global move_thread_flag_1362=0
    thread move_thread_1362():
      enter_critical
      move_thread_flag_1362 = 1
      local towardsPos=calculate_point_to_move_towards(p[0.0,0.0,0.0,0.0,0.0,0.0], [0.0,0.0,-1.0], 1000.0)
      movel(towardsPos, a=0.007, v=0.007)
      move_thread_flag_1362 = 2
      exit_critical
    end
    move_thread_flag_1362 = 0
    move_thread_han_1362 = run move_thread_1362()
    while (True):
      local targetTcpDirection=get_target_tcp_speed()
      local stepsToRetract=tool_contact(direction=targetTcpDirection)
      if (stepsToRetract > 0):
        kill move_thread_han_1362
        stopl(0.007)
        local backTrackMovement=get_actual_joint_positions_history(stepsToRetract)
        local contactPose=get_forward_kin(backTrackMovement)
        local posDir=[targetTcpDirection[0],targetTcpDirection[1],targetTcpDirection[2]]
        local retractTo=contactPose
        if (norm(posDir) > 1e-6):
          local normalizedPosDir=normalize(posDir)
          local additionalRetraction=p[normalizedPosDir[0] * 0.0, normalizedPosDir[1] * 0.0, normalizedPosDir[2] * 0.0, 0, 0, 0]
          retractTo = pose_sub(contactPose, additionalRetraction)
        end
        movel(retractTo, a=0.007, v=0.1)
        $ 1363 "Until (tool_contact_detection)"
        break
      end
      sync()
    end
    $ 1364 "Direction: Base Z+"
    global move_thread_flag_1364=0
    thread move_thread_1364():
      enter_critical
      move_thread_flag_1364 = 1
      local towardsPos=calculate_point_to_move_towards(p[0.0,0.0,0.0,0.0,0.0,0.0], [0.0,0.0,1.0], 0.08)
      movel(towardsPos, a=0.15, v=0.1)
      move_thread_flag_1364 = 2
      exit_critical
    end
    move_thread_flag_1364 = 0
    move_thread_han_1364 = run move_thread_1364()
    while (True):
      sleep(1.0E-10)
      if (move_thread_flag_1364 > 1):
        join move_thread_han_1364
        $ 1365 "Until (distance)"
        break
      end
      sync()
    end
    $ 1366 "Linea9_B" "breakAfter"
    movel(Linea9_B_p, a=0.5, v=0.1)
    $ 1367 "bajada_comprobacion"
    $ 1368 "Direction: Base Z-"
    global move_thread_flag_1368=0
    thread move_thread_1368():
      enter_critical
      move_thread_flag_1368 = 1
      local towardsPos=calculate_point_to_move_towards(p[0.0,0.0,0.0,0.0,0.0,0.0], [0.0,0.0,-1.0], 0.071)
      movel(towardsPos, a=0.15, v=0.1)
      move_thread_flag_1368 = 2
      exit_critical
    end
    move_thread_flag_1368 = 0
    move_thread_han_1368 = run move_thread_1368()
    while (True):
      sleep(1.0E-10)
      if (move_thread_flag_1368 > 1):
        join move_thread_han_1368
        $ 1369 "Until (distance)"
        break
      end
      sync()
    end
    $ 1370 "Direction: Base Z-"
    global move_thread_flag_1370=0
    thread move_thread_1370():
      enter_critical
      move_thread_flag_1370 = 1
      local towardsPos=calculate_point_to_move_towards(p[0.0,0.0,0.0,0.0,0.0,0.0], [0.0,0.0,-1.0], 1000.0)
      movel(towardsPos, a=0.007, v=0.007)
      move_thread_flag_1370 = 2
      exit_critical
    end
    move_thread_flag_1370 = 0
    move_thread_han_1370 = run move_thread_1370()
    while (True):
      local targetTcpDirection=get_target_tcp_speed()
      local stepsToRetract=tool_contact(direction=targetTcpDirection)
      if (stepsToRetract > 0):
        kill move_thread_han_1370
        stopl(0.007)
        local backTrackMovement=get_actual_joint_positions_history(stepsToRetract)
        local contactPose=get_forward_kin(backTrackMovement)
        local posDir=[targetTcpDirection[0],targetTcpDirection[1],targetTcpDirection[2]]
        local retractTo=contactPose
        if (norm(posDir) > 1e-6):
          local normalizedPosDir=normalize(posDir)
          local additionalRetraction=p[normalizedPosDir[0] * 0.0, normalizedPosDir[1] * 0.0, normalizedPosDir[2] * 0.0, 0, 0, 0]
          retractTo = pose_sub(contactPose, additionalRetraction)
        end
        movel(retractTo, a=0.007, v=0.1)
        $ 1371 "Until (tool_contact_detection)"
        break
      end
      sync()
    end
    $ 1372 "Direction: Base Z+"
    global move_thread_flag_1372=0
    thread move_thread_1372():
      enter_critical
      move_thread_flag_1372 = 1
      local towardsPos=calculate_point_to_move_towards(p[0.0,0.0,0.0,0.0,0.0,0.0], [0.0,0.0,1.0], 0.08)
      movel(towardsPos, a=0.15, v=0.1)
      move_thread_flag_1372 = 2
      exit_critical
    end
    move_thread_flag_1372 = 0
    move_thread_han_1372 = run move_thread_1372()
    while (True):
      sleep(1.0E-10)
      if (move_thread_flag_1372 > 1):
        join move_thread_han_1372
        $ 1373 "Until (distance)"
        break
      end
      sync()
    end
    $ 1374 "AB"
    $ 1375 "'desbaste_inicial'"
    # 'desbaste_inicial'
    $ 1376 "bajada_broca≔p[0,0,-0.008,0,0,0]"
    global bajada_broca=p[0,0,-0.008,0,0,0]
    $ 1377 "barrenos_menos1≔2"
    global barrenos_menos1=2
    $ 1378 "barreno_actual≔2"
    global barreno_actual=2
    $ 1379 "Loop barreno_actual≤barrenos_menos1"
    while (barreno_actual <= barrenos_menos1):
      $ 1380 "Perforacion"
      $ 1381 "MoveL"
      $ 1382 "internos≔interpolate_pose(Linea9_A, Linea9_B, barreno_actual/barrenos_menos1)"
      global internos= interpolate_pose (Linea9_A_p, Linea9_B_p, barreno_actual/barrenos_menos1)
      $ 1383 "internos" "breakAfter"
      movel(internos, a=0.5, v=0.1)
      $ 1384 "'desbaste_inicial'"
      # 'desbaste_inicial'
      $ 1385 "bajada_broca≔p[0,0,-0.024,0,0,0]"
      global bajada_broca=p[0,0,-0.024,0,0,0]
      $ 1386 "bajada≔p[0,0,0.024,0,0,0]"
      global bajada=p[0,0,0.024,0,0,0]
      $ 1387 "Direction: Base Z-"
      global move_thread_flag_1387=0
      thread move_thread_1387():
        enter_critical
        move_thread_flag_1387 = 1
        local towardsPos=calculate_point_to_move_towards(p[0.0,0.0,0.0,0.0,0.0,0.0], [0.0,0.0,-1.0], 0.071)
        movel(towardsPos, a=0.15, v=0.1)
        move_thread_flag_1387 = 2
        exit_critical
      end
      move_thread_flag_1387 = 0
      move_thread_han_1387 = run move_thread_1387()
      while (True):
        sleep(1.0E-10)
        if (move_thread_flag_1387 > 1):
          join move_thread_han_1387
          $ 1388 "Until (distance)"
          break
        end
        sync()
      end
      $ 1389 "Direction: Base Z-"
      global move_thread_flag_1389=0
      thread move_thread_1389():
        enter_critical
        move_thread_flag_1389 = 1
        local towardsPos=calculate_point_to_move_towards(p[0.0,0.0,0.0,0.0,0.0,0.0], [0.0,0.0,-1.0], 1000.0)
        movel(towardsPos, a=0.01, v=0.01)
        move_thread_flag_1389 = 2
        exit_critical
      end
      move_thread_flag_1389 = 0
      move_thread_han_1389 = run move_thread_1389()
      while (True):
        local targetTcpDirection=get_target_tcp_speed()
        local stepsToRetract=tool_contact(direction=targetTcpDirection)
        if (stepsToRetract > 0):
          kill move_thread_han_1389
          stopl(0.01)
          local backTrackMovement=get_actual_joint_positions_history(stepsToRetract)
          local contactPose=get_forward_kin(backTrackMovement)
          local posDir=[targetTcpDirection[0],targetTcpDirection[1],targetTcpDirection[2]]
          local retractTo=contactPose
          if (norm(posDir) > 1e-6):
            local normalizedPosDir=normalize(posDir)
            local additionalRetraction=p[normalizedPosDir[0] * 0.0, normalizedPosDir[1] * 0.0, normalizedPosDir[2] * 0.0, 0, 0, 0]
            retractTo = pose_sub(contactPose, additionalRetraction)
          end
          movel(retractTo, a=0.01, v=0.1)
          $ 1390 "Until (tool_contact_detection)"
          break
        end
        sync()
      end
      $ 1391 "Popup: punto contacto alanzdo"
      popup("punto contacto alanzdo", "Mensaje", False, False, blocking=True)
      $ 1392 "Direction: Base Z+"
      global move_thread_flag_1392=0
      thread move_thread_1392():
        enter_critical
        move_thread_flag_1392 = 1
        local towardsPos=calculate_point_to_move_towards(p[0.0,0.0,0.0,0.0,0.0,0.0], [0.0,0.0,1.0], 0.007)
        movel(towardsPos, a=0.015, v=0.015)
        move_thread_flag_1392 = 2
        exit_critical
      end
      move_thread_flag_1392 = 0
      move_thread_han_1392 = run move_thread_1392()
      while (True):
        sleep(1.0E-10)
        if (move_thread_flag_1392 > 1):
          join move_thread_han_1392
          $ 1393 "Until (distance)"
          break
        end
        sync()
      end
      $ 1394 "Wait: 0.3"
      sleep(0.3)
      $ 1395 "Set CO[1]=Encender"
      set_configurable_digital_out(1, True)
      $ 1396 "Wait: 0.3"
      sleep(0.3)
      $ 1397 "Loop 1 times"
      Loop_114 = 0
      while (Loop_114 < 1):
        $ 1398 "bajar≔pose_add(get_actual_tcp_pose(), bajada_broca)"
        global bajar= pose_add ( get_actual_tcp_pose (), bajada_broca)
        $ 1399 "bajar" "breakAfter"
        movel(bajar, a=0.01, v=0.01)
        $ 1400 "subir≔pose_sub(get_actual_tcp_pose(), bajada_broca)"
        global subir= pose_sub ( get_actual_tcp_pose (), bajada_broca)
        $ 1401 "Direction: Base Z+"
        global move_thread_flag_1401=0
        thread move_thread_1401():
          enter_critical
          move_thread_flag_1401 = 1
          local towardsPos=calculate_point_to_move_towards(p[0.0,0.0,0.0,0.0,0.0,0.0], [0.0,0.0,1.0], 0.002)
          movel(towardsPos, a=0.5, v=0.1)
          move_thread_flag_1401 = 2
          exit_critical
        end
        move_thread_flag_1401 = 0
        move_thread_han_1401 = run move_thread_1401()
        while (True):
          sleep(1.0E-10)
          if (move_thread_flag_1401 > 1):
            join move_thread_han_1401
            $ 1402 "Until (distance)"
            break
          end
          sync()
        end
        $ 1403 "Set CO[1]=Apagar"
        set_configurable_digital_out(1, False)
        $ 1404 "subir" "breakAfter"
        movel(subir, a=0.015, v=0.015)
        $ 1405 "bajada_broca≔pose_sub(bajada_broca, bajada)"
        global bajada_broca= pose_sub (bajada_broca, bajada)
        Loop_114 = Loop_114 + 1
      end
      $ 1406 "Direction: Base Z+"
      global move_thread_flag_1406=0
      thread move_thread_1406():
        enter_critical
        move_thread_flag_1406 = 1
        local towardsPos=calculate_point_to_move_towards(p[0.0,0.0,0.0,0.0,0.0,0.0], [0.0,0.0,1.0], 0.08)
        movel(towardsPos, a=0.15, v=0.1)
        move_thread_flag_1406 = 2
        exit_critical
      end
      move_thread_flag_1406 = 0
      move_thread_han_1406 = run move_thread_1406()
      while (True):
        sleep(1.0E-10)
        if (move_thread_flag_1406 > 1):
          join move_thread_han_1406
          $ 1407 "Until (distance)"
          break
        end
        sync()
      end
      $ 1408 "Set CO[1]=Apagar"
      set_configurable_digital_out(1, False)
      $ 1409 "barreno_actual≔barreno_actual+1"
      global barreno_actual=barreno_actual+1
      $ 1410 "Call Quitar_broca"
      Quitar_broca()
      $ 1411 "Call Poner_broca"
      Poner_broca()
    end
    $ 1412 "Popup: Linea9 con chica Terminada!"
    popup("Linea9 con chica Terminada!", "Mensaje", False, False, blocking=True)
    $ 1413 "Linea10"
    $ 1414 "Marcar_puntos"
    $ 1415 "MoveL"
    $ 1416 "Home2" "breakAfter"
    movel(Home2_p, a=0.5, v=0.1)
    $ 1417 "Linea10_A" "breakAfter"
    movel(Linea10_A_p, a=0.5, v=0.1)
    $ 1418 "bajada_comprobacion"
    $ 1419 "Direction: Base Z-"
    global move_thread_flag_1419=0
    thread move_thread_1419():
      enter_critical
      move_thread_flag_1419 = 1
      local towardsPos=calculate_point_to_move_towards(p[0.0,0.0,0.0,0.0,0.0,0.0], [0.0,0.0,-1.0], 0.071)
      movel(towardsPos, a=0.15, v=0.1)
      move_thread_flag_1419 = 2
      exit_critical
    end
    move_thread_flag_1419 = 0
    move_thread_han_1419 = run move_thread_1419()
    while (True):
      sleep(1.0E-10)
      if (move_thread_flag_1419 > 1):
        join move_thread_han_1419
        $ 1420 "Until (distance)"
        break
      end
      sync()
    end
    $ 1421 "Direction: Base Z-"
    global move_thread_flag_1421=0
    thread move_thread_1421():
      enter_critical
      move_thread_flag_1421 = 1
      local towardsPos=calculate_point_to_move_towards(p[0.0,0.0,0.0,0.0,0.0,0.0], [0.0,0.0,-1.0], 1000.0)
      movel(towardsPos, a=0.007, v=0.007)
      move_thread_flag_1421 = 2
      exit_critical
    end
    move_thread_flag_1421 = 0
    move_thread_han_1421 = run move_thread_1421()
    while (True):
      local targetTcpDirection=get_target_tcp_speed()
      local stepsToRetract=tool_contact(direction=targetTcpDirection)
      if (stepsToRetract > 0):
        kill move_thread_han_1421
        stopl(0.02)
        local backTrackMovement=get_actual_joint_positions_history(stepsToRetract)
        local contactPose=get_forward_kin(backTrackMovement)
        local posDir=[targetTcpDirection[0],targetTcpDirection[1],targetTcpDirection[2]]
        local retractTo=contactPose
        if (norm(posDir) > 1e-6):
          local normalizedPosDir=normalize(posDir)
          local additionalRetraction=p[normalizedPosDir[0] * 0.0, normalizedPosDir[1] * 0.0, normalizedPosDir[2] * 0.0, 0, 0, 0]
          retractTo = pose_sub(contactPose, additionalRetraction)
        end
        movel(retractTo, a=0.02, v=0.1)
        $ 1422 "Until (tool_contact_detection)"
        break
      end
      sync()
    end
    $ 1423 "Direction: Base Z+"
    global move_thread_flag_1423=0
    thread move_thread_1423():
      enter_critical
      move_thread_flag_1423 = 1
      local towardsPos=calculate_point_to_move_towards(p[0.0,0.0,0.0,0.0,0.0,0.0], [0.0,0.0,1.0], 0.08)
      movel(towardsPos, a=0.15, v=0.1)
      move_thread_flag_1423 = 2
      exit_critical
    end
    move_thread_flag_1423 = 0
    move_thread_han_1423 = run move_thread_1423()
    while (True):
      sleep(1.0E-10)
      if (move_thread_flag_1423 > 1):
        join move_thread_han_1423
        $ 1424 "Until (distance)"
        break
      end
      sync()
    end
    $ 1425 "Linea10_B" "breakAfter"
    movel(Linea10_B_p, a=0.5, v=0.1)
    $ 1426 "bajada_comprobacion"
    $ 1427 "Direction: Base Z-"
    global move_thread_flag_1427=0
    thread move_thread_1427():
      enter_critical
      move_thread_flag_1427 = 1
      local towardsPos=calculate_point_to_move_towards(p[0.0,0.0,0.0,0.0,0.0,0.0], [0.0,0.0,-1.0], 0.071)
      movel(towardsPos, a=0.15, v=0.1)
      move_thread_flag_1427 = 2
      exit_critical
    end
    move_thread_flag_1427 = 0
    move_thread_han_1427 = run move_thread_1427()
    while (True):
      sleep(1.0E-10)
      if (move_thread_flag_1427 > 1):
        join move_thread_han_1427
        $ 1428 "Until (distance)"
        break
      end
      sync()
    end
    $ 1429 "Direction: Base Z-"
    global move_thread_flag_1429=0
    thread move_thread_1429():
      enter_critical
      move_thread_flag_1429 = 1
      local towardsPos=calculate_point_to_move_towards(p[0.0,0.0,0.0,0.0,0.0,0.0], [0.0,0.0,-1.0], 1000.0)
      movel(towardsPos, a=0.007, v=0.007)
      move_thread_flag_1429 = 2
      exit_critical
    end
    move_thread_flag_1429 = 0
    move_thread_han_1429 = run move_thread_1429()
    while (True):
      local targetTcpDirection=get_target_tcp_speed()
      local stepsToRetract=tool_contact(direction=targetTcpDirection)
      if (stepsToRetract > 0):
        kill move_thread_han_1429
        stopl(0.02)
        local backTrackMovement=get_actual_joint_positions_history(stepsToRetract)
        local contactPose=get_forward_kin(backTrackMovement)
        local posDir=[targetTcpDirection[0],targetTcpDirection[1],targetTcpDirection[2]]
        local retractTo=contactPose
        if (norm(posDir) > 1e-6):
          local normalizedPosDir=normalize(posDir)
          local additionalRetraction=p[normalizedPosDir[0] * 0.0, normalizedPosDir[1] * 0.0, normalizedPosDir[2] * 0.0, 0, 0, 0]
          retractTo = pose_sub(contactPose, additionalRetraction)
        end
        movel(retractTo, a=0.02, v=0.1)
        $ 1430 "Until (tool_contact_detection)"
        break
      end
      sync()
    end
    $ 1431 "Direction: Base Z+"
    global move_thread_flag_1431=0
    thread move_thread_1431():
      enter_critical
      move_thread_flag_1431 = 1
      local towardsPos=calculate_point_to_move_towards(p[0.0,0.0,0.0,0.0,0.0,0.0], [0.0,0.0,1.0], 0.08)
      movel(towardsPos, a=0.15, v=0.1)
      move_thread_flag_1431 = 2
      exit_critical
    end
    move_thread_flag_1431 = 0
    move_thread_han_1431 = run move_thread_1431()
    while (True):
      sleep(1.0E-10)
      if (move_thread_flag_1431 > 1):
        join move_thread_han_1431
        $ 1432 "Until (distance)"
        break
      end
      sync()
    end
    $ 1433 "AB"
    $ 1434 "'desbaste_inicial'"
    # 'desbaste_inicial'
    $ 1435 "bajada_broca≔p[0,0,-0.008,0,0,0]"
    global bajada_broca=p[0,0,-0.008,0,0,0]
    $ 1436 "barrenos_menos1≔2"
    global barrenos_menos1=2
    $ 1437 "barreno_actual≔0"
    global barreno_actual=0
    $ 1438 "Loop barreno_actual≤barrenos_menos1"
    while (barreno_actual <= barrenos_menos1):
      $ 1439 "Perforacion"
      $ 1440 "MoveL"
      $ 1441 "internos≔interpolate_pose(Linea10_A, Linea10_B, barreno_actual/barrenos_menos1)"
      global internos= interpolate_pose (Linea10_A_p, Linea10_B_p, barreno_actual/barrenos_menos1)
      $ 1442 "internos" "breakAfter"
      movel(internos, a=0.5, v=0.1)
      $ 1443 "'desbaste_inicial'"
      # 'desbaste_inicial'
      $ 1444 "bajada_broca≔p[0,0,-0.024,0,0,0]"
      global bajada_broca=p[0,0,-0.024,0,0,0]
      $ 1445 "bajada≔p[0,0,0.024,0,0,0]"
      global bajada=p[0,0,0.024,0,0,0]
      $ 1446 "Direction: Base Z-"
      global move_thread_flag_1446=0
      thread move_thread_1446():
        enter_critical
        move_thread_flag_1446 = 1
        local towardsPos=calculate_point_to_move_towards(p[0.0,0.0,0.0,0.0,0.0,0.0], [0.0,0.0,-1.0], 0.071)
        movel(towardsPos, a=0.15, v=0.1)
        move_thread_flag_1446 = 2
        exit_critical
      end
      move_thread_flag_1446 = 0
      move_thread_han_1446 = run move_thread_1446()
      while (True):
        sleep(1.0E-10)
        if (move_thread_flag_1446 > 1):
          join move_thread_han_1446
          $ 1447 "Until (distance)"
          break
        end
        sync()
      end
      $ 1448 "Direction: Base Z-"
      global move_thread_flag_1448=0
      thread move_thread_1448():
        enter_critical
        move_thread_flag_1448 = 1
        local towardsPos=calculate_point_to_move_towards(p[0.0,0.0,0.0,0.0,0.0,0.0], [0.0,0.0,-1.0], 1000.0)
        movel(towardsPos, a=0.007, v=0.007)
        move_thread_flag_1448 = 2
        exit_critical
      end
      move_thread_flag_1448 = 0
      move_thread_han_1448 = run move_thread_1448()
      while (True):
        local targetTcpDirection=get_target_tcp_speed()
        local stepsToRetract=tool_contact(direction=targetTcpDirection)
        if (stepsToRetract > 0):
          kill move_thread_han_1448
          stopl(0.02)
          local backTrackMovement=get_actual_joint_positions_history(stepsToRetract)
          local contactPose=get_forward_kin(backTrackMovement)
          local posDir=[targetTcpDirection[0],targetTcpDirection[1],targetTcpDirection[2]]
          local retractTo=contactPose
          if (norm(posDir) > 1e-6):
            local normalizedPosDir=normalize(posDir)
            local additionalRetraction=p[normalizedPosDir[0] * 0.0, normalizedPosDir[1] * 0.0, normalizedPosDir[2] * 0.0, 0, 0, 0]
            retractTo = pose_sub(contactPose, additionalRetraction)
          end
          movel(retractTo, a=0.02, v=0.1)
          $ 1449 "Until (tool_contact_detection)"
          break
        end
        sync()
      end
      $ 1450 "Popup: punto contacto alanzdo"
      popup("punto contacto alanzdo", "Mensaje", False, False, blocking=True)
      $ 1451 "Direction: Base Z+"
      global move_thread_flag_1451=0
      thread move_thread_1451():
        enter_critical
        move_thread_flag_1451 = 1
        local towardsPos=calculate_point_to_move_towards(p[0.0,0.0,0.0,0.0,0.0,0.0], [0.0,0.0,1.0], 0.007)
        movel(towardsPos, a=0.015, v=0.015)
        move_thread_flag_1451 = 2
        exit_critical
      end
      move_thread_flag_1451 = 0
      move_thread_han_1451 = run move_thread_1451()
      while (True):
        sleep(1.0E-10)
        if (move_thread_flag_1451 > 1):
          join move_thread_han_1451
          $ 1452 "Until (distance)"
          break
        end
        sync()
      end
      $ 1453 "Wait: 0.3"
      sleep(0.3)
      $ 1454 "Set CO[1]=Encender"
      set_configurable_digital_out(1, True)
      $ 1455 "Wait: 0.3"
      sleep(0.3)
      $ 1456 "Loop 1 times"
      Loop_118 = 0
      while (Loop_118 < 1):
        $ 1457 "bajar≔pose_add(get_actual_tcp_pose(), bajada_broca)"
        global bajar= pose_add ( get_actual_tcp_pose (), bajada_broca)
        $ 1458 "bajar" "breakAfter"
        movel(bajar, a=0.004, v=0.004)
        $ 1459 "subir≔pose_sub(get_actual_tcp_pose(), bajada_broca)"
        global subir= pose_sub ( get_actual_tcp_pose (), bajada_broca)
        $ 1460 "Direction: Base Z+"
        global move_thread_flag_1460=0
        thread move_thread_1460():
          enter_critical
          move_thread_flag_1460 = 1
          local towardsPos=calculate_point_to_move_towards(p[0.0,0.0,0.0,0.0,0.0,0.0], [0.0,0.0,1.0], 0.002)
          movel(towardsPos, a=0.015, v=0.015)
          move_thread_flag_1460 = 2
          exit_critical
        end
        move_thread_flag_1460 = 0
        move_thread_han_1460 = run move_thread_1460()
        while (True):
          sleep(1.0E-10)
          if (move_thread_flag_1460 > 1):
            join move_thread_han_1460
            $ 1461 "Until (distance)"
            break
          end
          sync()
        end
        $ 1462 "Set CO[1]=Apagar"
        set_configurable_digital_out(1, False)
        $ 1463 "subir" "breakAfter"
        movel(subir, a=0.015, v=0.015)
        $ 1464 "bajada_broca≔pose_sub(bajada_broca, bajada)"
        global bajada_broca= pose_sub (bajada_broca, bajada)
        Loop_118 = Loop_118 + 1
      end
      $ 1465 "Direction: Base Z+"
      global move_thread_flag_1465=0
      thread move_thread_1465():
        enter_critical
        move_thread_flag_1465 = 1
        local towardsPos=calculate_point_to_move_towards(p[0.0,0.0,0.0,0.0,0.0,0.0], [0.0,0.0,1.0], 0.08)
        movel(towardsPos, a=0.15, v=0.1)
        move_thread_flag_1465 = 2
        exit_critical
      end
      move_thread_flag_1465 = 0
      move_thread_han_1465 = run move_thread_1465()
      while (True):
        sleep(1.0E-10)
        if (move_thread_flag_1465 > 1):
          join move_thread_han_1465
          $ 1466 "Until (distance)"
          break
        end
        sync()
      end
      $ 1467 "Set CO[1]=Apagar"
      set_configurable_digital_out(1, False)
      $ 1468 "barreno_actual≔barreno_actual+1"
      global barreno_actual=barreno_actual+1
    end
    $ 1471 "Popup: Linea10 con chica Terminada!"
    popup("Linea10 con chica Terminada!", "Mensaje", False, False, blocking=True)
    $ 1472 "Linea11"
    $ 1473 "Marcar_puntos"
    $ 1474 "MoveL"
    $ 1475 "Linea11_A" "breakAfter"
    movel(Linea11_A_p, a=0.5, v=0.1)
    $ 1476 "bajada_comprobacion"
    $ 1477 "Direction: Base Z-"
    global move_thread_flag_1477=0
    thread move_thread_1477():
      enter_critical
      move_thread_flag_1477 = 1
      local towardsPos=calculate_point_to_move_towards(p[0.0,0.0,0.0,0.0,0.0,0.0], [0.0,0.0,-1.0], 0.071)
      movel(towardsPos, a=0.15, v=0.1)
      move_thread_flag_1477 = 2
      exit_critical
    end
    move_thread_flag_1477 = 0
    move_thread_han_1477 = run move_thread_1477()
    while (True):
      sleep(1.0E-10)
      if (move_thread_flag_1477 > 1):
        join move_thread_han_1477
        $ 1478 "Until (distance)"
        break
      end
      sync()
    end
    $ 1479 "Direction: Base Z-"
    global move_thread_flag_1479=0
    thread move_thread_1479():
      enter_critical
      move_thread_flag_1479 = 1
      local towardsPos=calculate_point_to_move_towards(p[0.0,0.0,0.0,0.0,0.0,0.0], [0.0,0.0,-1.0], 1000.0)
      movel(towardsPos, a=0.007, v=0.007)
      move_thread_flag_1479 = 2
      exit_critical
    end
    move_thread_flag_1479 = 0
    move_thread_han_1479 = run move_thread_1479()
    while (True):
      local targetTcpDirection=get_target_tcp_speed()
      local stepsToRetract=tool_contact(direction=targetTcpDirection)
      if (stepsToRetract > 0):
        kill move_thread_han_1479
        stopl(0.02)
        local backTrackMovement=get_actual_joint_positions_history(stepsToRetract)
        local contactPose=get_forward_kin(backTrackMovement)
        local posDir=[targetTcpDirection[0],targetTcpDirection[1],targetTcpDirection[2]]
        local retractTo=contactPose
        if (norm(posDir) > 1e-6):
          local normalizedPosDir=normalize(posDir)
          local additionalRetraction=p[normalizedPosDir[0] * 0.0, normalizedPosDir[1] * 0.0, normalizedPosDir[2] * 0.0, 0, 0, 0]
          retractTo = pose_sub(contactPose, additionalRetraction)
        end
        movel(retractTo, a=0.02, v=0.1)
        $ 1480 "Until (tool_contact_detection)"
        break
      end
      sync()
    end
    $ 1481 "Direction: Base Z+"
    global move_thread_flag_1481=0
    thread move_thread_1481():
      enter_critical
      move_thread_flag_1481 = 1
      local towardsPos=calculate_point_to_move_towards(p[0.0,0.0,0.0,0.0,0.0,0.0], [0.0,0.0,1.0], 0.08)
      movel(towardsPos, a=0.15, v=0.1)
      move_thread_flag_1481 = 2
      exit_critical
    end
    move_thread_flag_1481 = 0
    move_thread_han_1481 = run move_thread_1481()
    while (True):
      sleep(1.0E-10)
      if (move_thread_flag_1481 > 1):
        join move_thread_han_1481
        $ 1482 "Until (distance)"
        break
      end
      sync()
    end
    $ 1483 "Linea11_B" "breakAfter"
    movel(Linea11_B_p, a=0.5, v=0.1)
    $ 1484 "bajada_comprobacion"
    $ 1485 "Direction: Base Z-"
    global move_thread_flag_1485=0
    thread move_thread_1485():
      enter_critical
      move_thread_flag_1485 = 1
      local towardsPos=calculate_point_to_move_towards(p[0.0,0.0,0.0,0.0,0.0,0.0], [0.0,0.0,-1.0], 0.071)
      movel(towardsPos, a=0.15, v=0.1)
      move_thread_flag_1485 = 2
      exit_critical
    end
    move_thread_flag_1485 = 0
    move_thread_han_1485 = run move_thread_1485()
    while (True):
      sleep(1.0E-10)
      if (move_thread_flag_1485 > 1):
        join move_thread_han_1485
        $ 1486 "Until (distance)"
        break
      end
      sync()
    end
    $ 1487 "Direction: Base Z-"
    global move_thread_flag_1487=0
    thread move_thread_1487():
      enter_critical
      move_thread_flag_1487 = 1
      local towardsPos=calculate_point_to_move_towards(p[0.0,0.0,0.0,0.0,0.0,0.0], [0.0,0.0,-1.0], 1000.0)
      movel(towardsPos, a=0.007, v=0.007)
      move_thread_flag_1487 = 2
      exit_critical
    end
    move_thread_flag_1487 = 0
    move_thread_han_1487 = run move_thread_1487()
    while (True):
      local targetTcpDirection=get_target_tcp_speed()
      local stepsToRetract=tool_contact(direction=targetTcpDirection)
      if (stepsToRetract > 0):
        kill move_thread_han_1487
        stopl(0.02)
        local backTrackMovement=get_actual_joint_positions_history(stepsToRetract)
        local contactPose=get_forward_kin(backTrackMovement)
        local posDir=[targetTcpDirection[0],targetTcpDirection[1],targetTcpDirection[2]]
        local retractTo=contactPose
        if (norm(posDir) > 1e-6):
          local normalizedPosDir=normalize(posDir)
          local additionalRetraction=p[normalizedPosDir[0] * 0.0, normalizedPosDir[1] * 0.0, normalizedPosDir[2] * 0.0, 0, 0, 0]
          retractTo = pose_sub(contactPose, additionalRetraction)
        end
        movel(retractTo, a=0.02, v=0.1)
        $ 1488 "Until (tool_contact_detection)"
        break
      end
      sync()
    end
    $ 1489 "Direction: Base Z+"
    global move_thread_flag_1489=0
    thread move_thread_1489():
      enter_critical
      move_thread_flag_1489 = 1
      local towardsPos=calculate_point_to_move_towards(p[0.0,0.0,0.0,0.0,0.0,0.0], [0.0,0.0,1.0], 0.08)
      movel(towardsPos, a=0.15, v=0.1)
      move_thread_flag_1489 = 2
      exit_critical
    end
    move_thread_flag_1489 = 0
    move_thread_han_1489 = run move_thread_1489()
    while (True):
      sleep(1.0E-10)
      if (move_thread_flag_1489 > 1):
        join move_thread_han_1489
        $ 1490 "Until (distance)"
        break
      end
      sync()
    end
    $ 1491 "AB"
    $ 1492 "'desbaste_inicial'"
    # 'desbaste_inicial'
    $ 1493 "bajada_broca≔p[0,0,-0.008,0,0,0]"
    global bajada_broca=p[0,0,-0.008,0,0,0]
    $ 1494 "barrenos_menos1≔2"
    global barrenos_menos1=2
    $ 1495 "barreno_actual≔0"
    global barreno_actual=0
    $ 1496 "Loop barreno_actual≤barrenos_menos1"
    while (barreno_actual <= barrenos_menos1):
      $ 1497 "Perforacion"
      $ 1498 "MoveL"
      $ 1501 "internos≔interpolate_pose(Linea11_A, Linea11_B, barreno_actual/barrenos_menos1)"
      global internos= interpolate_pose (Linea11_A_p, Linea11_B_p, barreno_actual/barrenos_menos1)
      $ 1502 "internos" "breakAfter"
      movel(internos, a=0.5, v=0.1)
      $ 1503 "'desbaste_inicial'"
      # 'desbaste_inicial'
      $ 1504 "bajada_broca≔p[0,0,-0.024,0,0,0]"
      global bajada_broca=p[0,0,-0.024,0,0,0]
      $ 1505 "bajada≔p[0,0,0.024,0,0,0]"
      global bajada=p[0,0,0.024,0,0,0]
      $ 1506 "Direction: Base Z-"
      global move_thread_flag_1506=0
      thread move_thread_1506():
        enter_critical
        move_thread_flag_1506 = 1
        local towardsPos=calculate_point_to_move_towards(p[0.0,0.0,0.0,0.0,0.0,0.0], [0.0,0.0,-1.0], 0.071)
        movel(towardsPos, a=0.15, v=0.1)
        move_thread_flag_1506 = 2
        exit_critical
      end
      move_thread_flag_1506 = 0
      move_thread_han_1506 = run move_thread_1506()
      while (True):
        sleep(1.0E-10)
        if (move_thread_flag_1506 > 1):
          join move_thread_han_1506
          $ 1507 "Until (distance)"
          break
        end
        sync()
      end
      $ 1508 "Direction: Base Z-"
      global move_thread_flag_1508=0
      thread move_thread_1508():
        enter_critical
        move_thread_flag_1508 = 1
        local towardsPos=calculate_point_to_move_towards(p[0.0,0.0,0.0,0.0,0.0,0.0], [0.0,0.0,-1.0], 1000.0)
        movel(towardsPos, a=0.007, v=0.007)
        move_thread_flag_1508 = 2
        exit_critical
      end
      move_thread_flag_1508 = 0
      move_thread_han_1508 = run move_thread_1508()
      while (True):
        local targetTcpDirection=get_target_tcp_speed()
        local stepsToRetract=tool_contact(direction=targetTcpDirection)
        if (stepsToRetract > 0):
          kill move_thread_han_1508
          stopl(0.02)
          local backTrackMovement=get_actual_joint_positions_history(stepsToRetract)
          local contactPose=get_forward_kin(backTrackMovement)
          local posDir=[targetTcpDirection[0],targetTcpDirection[1],targetTcpDirection[2]]
          local retractTo=contactPose
          if (norm(posDir) > 1e-6):
            local normalizedPosDir=normalize(posDir)
            local additionalRetraction=p[normalizedPosDir[0] * 0.0, normalizedPosDir[1] * 0.0, normalizedPosDir[2] * 0.0, 0, 0, 0]
            retractTo = pose_sub(contactPose, additionalRetraction)
          end
          movel(retractTo, a=0.02, v=0.1)
          $ 1509 "Until (tool_contact_detection)"
          break
        end
        sync()
      end
      $ 1510 "Popup: punto contacto alanzdo"
      popup("punto contacto alanzdo", "Mensaje", False, False, blocking=True)
      $ 1511 "Direction: Base Z+"
      global move_thread_flag_1511=0
      thread move_thread_1511():
        enter_critical
        move_thread_flag_1511 = 1
        local towardsPos=calculate_point_to_move_towards(p[0.0,0.0,0.0,0.0,0.0,0.0], [0.0,0.0,1.0], 0.007)
        movel(towardsPos, a=0.015, v=0.015)
        move_thread_flag_1511 = 2
        exit_critical
      end
      move_thread_flag_1511 = 0
      move_thread_han_1511 = run move_thread_1511()
      while (True):
        sleep(1.0E-10)
        if (move_thread_flag_1511 > 1):
          join move_thread_han_1511
          $ 1512 "Until (distance)"
          break
        end
        sync()
      end
      $ 1513 "Wait: 0.3"
      sleep(0.3)
      $ 1514 "Set CO[1]=Encender"
      set_configurable_digital_out(1, True)
      $ 1515 "Wait: 0.3"
      sleep(0.3)
      $ 1516 "Loop 1 times"
      Loop_122 = 0
      while (Loop_122 < 1):
        $ 1517 "bajar≔pose_add(get_actual_tcp_pose(), bajada_broca)"
        global bajar= pose_add ( get_actual_tcp_pose (), bajada_broca)
        $ 1518 "bajar" "breakAfter"
        movel(bajar, a=0.004, v=0.004)
        $ 1519 "subir≔pose_sub(get_actual_tcp_pose(), bajada_broca)"
        global subir= pose_sub ( get_actual_tcp_pose (), bajada_broca)
        $ 1520 "Direction: Base Z+"
        global move_thread_flag_1520=0
        thread move_thread_1520():
          enter_critical
          move_thread_flag_1520 = 1
          local towardsPos=calculate_point_to_move_towards(p[0.0,0.0,0.0,0.0,0.0,0.0], [0.0,0.0,1.0], 0.002)
          movel(towardsPos, a=0.015, v=0.015)
          move_thread_flag_1520 = 2
          exit_critical
        end
        move_thread_flag_1520 = 0
        move_thread_han_1520 = run move_thread_1520()
        while (True):
          sleep(1.0E-10)
          if (move_thread_flag_1520 > 1):
            join move_thread_han_1520
            $ 1521 "Until (distance)"
            break
          end
          sync()
        end
        $ 1522 "Set CO[1]=Apagar"
        set_configurable_digital_out(1, False)
        $ 1523 "subir" "breakAfter"
        movel(subir, a=0.015, v=0.015)
        $ 1524 "bajada_broca≔pose_sub(bajada_broca, bajada)"
        global bajada_broca= pose_sub (bajada_broca, bajada)
        Loop_122 = Loop_122 + 1
      end
      $ 1525 "Direction: Base Z+"
      global move_thread_flag_1525=0
      thread move_thread_1525():
        enter_critical
        move_thread_flag_1525 = 1
        local towardsPos=calculate_point_to_move_towards(p[0.0,0.0,0.0,0.0,0.0,0.0], [0.0,0.0,1.0], 0.08)
        movel(towardsPos, a=0.15, v=0.1)
        move_thread_flag_1525 = 2
        exit_critical
      end
      move_thread_flag_1525 = 0
      move_thread_han_1525 = run move_thread_1525()
      while (True):
        sleep(1.0E-10)
        if (move_thread_flag_1525 > 1):
          join move_thread_han_1525
          $ 1526 "Until (distance)"
          break
        end
        sync()
      end
      $ 1527 "Set CO[1]=Apagar"
      set_configurable_digital_out(1, False)
      $ 1528 "barreno_actual≔barreno_actual+1"
      global barreno_actual=barreno_actual+1
    end
    $ 1531 "Popup: Linea11 con chica Terminada!"
    popup("Linea11 con chica Terminada!", "Mensaje", False, False, blocking=True)
    $ 1532 "Linea12"
    $ 1533 "Marcar_puntos"
    $ 1534 "MoveL"
    $ 1535 "Linea12_A" "breakAfter"
    movel(Linea12_A_p, a=0.5, v=0.1)
    $ 1536 "bajada_comprobacion"
    $ 1537 "Direction: Base Z-"
    global move_thread_flag_1537=0
    thread move_thread_1537():
      enter_critical
      move_thread_flag_1537 = 1
      local towardsPos=calculate_point_to_move_towards(p[0.0,0.0,0.0,0.0,0.0,0.0], [0.0,0.0,-1.0], 0.071)
      movel(towardsPos, a=0.15, v=0.1)
      move_thread_flag_1537 = 2
      exit_critical
    end
    move_thread_flag_1537 = 0
    move_thread_han_1537 = run move_thread_1537()
    while (True):
      sleep(1.0E-10)
      if (move_thread_flag_1537 > 1):
        join move_thread_han_1537
        $ 1538 "Until (distance)"
        break
      end
      sync()
    end
    $ 1539 "Direction: Base Z-"
    global move_thread_flag_1539=0
    thread move_thread_1539():
      enter_critical
      move_thread_flag_1539 = 1
      local towardsPos=calculate_point_to_move_towards(p[0.0,0.0,0.0,0.0,0.0,0.0], [0.0,0.0,-1.0], 1000.0)
      movel(towardsPos, a=0.007, v=0.007)
      move_thread_flag_1539 = 2
      exit_critical
    end
    move_thread_flag_1539 = 0
    move_thread_han_1539 = run move_thread_1539()
    while (True):
      local targetTcpDirection=get_target_tcp_speed()
      local stepsToRetract=tool_contact(direction=targetTcpDirection)
      if (stepsToRetract > 0):
        kill move_thread_han_1539
        stopl(0.02)
        local backTrackMovement=get_actual_joint_positions_history(stepsToRetract)
        local contactPose=get_forward_kin(backTrackMovement)
        local posDir=[targetTcpDirection[0],targetTcpDirection[1],targetTcpDirection[2]]
        local retractTo=contactPose
        if (norm(posDir) > 1e-6):
          local normalizedPosDir=normalize(posDir)
          local additionalRetraction=p[normalizedPosDir[0] * 0.0, normalizedPosDir[1] * 0.0, normalizedPosDir[2] * 0.0, 0, 0, 0]
          retractTo = pose_sub(contactPose, additionalRetraction)
        end
        movel(retractTo, a=0.02, v=0.1)
        $ 1540 "Until (tool_contact_detection)"
        break
      end
      sync()
    end
    $ 1541 "Direction: Base Z+"
    global move_thread_flag_1541=0
    thread move_thread_1541():
      enter_critical
      move_thread_flag_1541 = 1
      local towardsPos=calculate_point_to_move_towards(p[0.0,0.0,0.0,0.0,0.0,0.0], [0.0,0.0,1.0], 0.08)
      movel(towardsPos, a=0.15, v=0.1)
      move_thread_flag_1541 = 2
      exit_critical
    end
    move_thread_flag_1541 = 0
    move_thread_han_1541 = run move_thread_1541()
    while (True):
      sleep(1.0E-10)
      if (move_thread_flag_1541 > 1):
        join move_thread_han_1541
        $ 1542 "Until (distance)"
        break
      end
      sync()
    end
    $ 1543 "Linea12_B" "breakAfter"
    movel(Linea12_B_p, a=0.5, v=0.1)
    $ 1544 "bajada_comprobacion"
    $ 1545 "Direction: Base Z-"
    global move_thread_flag_1545=0
    thread move_thread_1545():
      enter_critical
      move_thread_flag_1545 = 1
      local towardsPos=calculate_point_to_move_towards(p[0.0,0.0,0.0,0.0,0.0,0.0], [0.0,0.0,-1.0], 0.071)
      movel(towardsPos, a=0.15, v=0.1)
      move_thread_flag_1545 = 2
      exit_critical
    end
    move_thread_flag_1545 = 0
    move_thread_han_1545 = run move_thread_1545()
    while (True):
      sleep(1.0E-10)
      if (move_thread_flag_1545 > 1):
        join move_thread_han_1545
        $ 1546 "Until (distance)"
        break
      end
      sync()
    end
    $ 1547 "Direction: Base Z-"
    global move_thread_flag_1547=0
    thread move_thread_1547():
      enter_critical
      move_thread_flag_1547 = 1
      local towardsPos=calculate_point_to_move_towards(p[0.0,0.0,0.0,0.0,0.0,0.0], [0.0,0.0,-1.0], 1000.0)
      movel(towardsPos, a=0.007, v=0.007)
      move_thread_flag_1547 = 2
      exit_critical
    end
    move_thread_flag_1547 = 0
    move_thread_han_1547 = run move_thread_1547()
    while (True):
      local targetTcpDirection=get_target_tcp_speed()
      local stepsToRetract=tool_contact(direction=targetTcpDirection)
      if (stepsToRetract > 0):
        kill move_thread_han_1547
        stopl(0.02)
        local backTrackMovement=get_actual_joint_positions_history(stepsToRetract)
        local contactPose=get_forward_kin(backTrackMovement)
        local posDir=[targetTcpDirection[0],targetTcpDirection[1],targetTcpDirection[2]]
        local retractTo=contactPose
        if (norm(posDir) > 1e-6):
          local normalizedPosDir=normalize(posDir)
          local additionalRetraction=p[normalizedPosDir[0] * 0.0, normalizedPosDir[1] * 0.0, normalizedPosDir[2] * 0.0, 0, 0, 0]
          retractTo = pose_sub(contactPose, additionalRetraction)
        end
        movel(retractTo, a=0.02, v=0.1)
        $ 1548 "Until (tool_contact_detection)"
        break
      end
      sync()
    end
    $ 1549 "Direction: Base Z+"
    global move_thread_flag_1549=0
    thread move_thread_1549():
      enter_critical
      move_thread_flag_1549 = 1
      local towardsPos=calculate_point_to_move_towards(p[0.0,0.0,0.0,0.0,0.0,0.0], [0.0,0.0,1.0], 0.08)
      movel(towardsPos, a=0.15, v=0.1)
      move_thread_flag_1549 = 2
      exit_critical
    end
    move_thread_flag_1549 = 0
    move_thread_han_1549 = run move_thread_1549()
    while (True):
      sleep(1.0E-10)
      if (move_thread_flag_1549 > 1):
        join move_thread_han_1549
        $ 1550 "Until (distance)"
        break
      end
      sync()
    end
    $ 1551 "AB"
    $ 1552 "'desbaste_inicial'"
    # 'desbaste_inicial'
    $ 1553 "bajada_broca≔p[0,0,-0.008,0,0,0]"
    global bajada_broca=p[0,0,-0.008,0,0,0]
    $ 1554 "barrenos_menos1≔7"
    global barrenos_menos1=7
    $ 1555 "barreno_actual≔0"
    global barreno_actual=0
    $ 1556 "Loop barreno_actual≤barrenos_menos1"
    while (barreno_actual <= barrenos_menos1):
      $ 1557 "Perforacion"
      $ 1558 "MoveL"
      $ 1559 "If barreno_actual≟2"
      if (barreno_actual == 2):
        $ 1560 "barreno_actual≔barreno_actual+1"
        global barreno_actual=barreno_actual+1
      end
      $ 1561 "internos≔interpolate_pose(Linea12_A, Linea12_B, barreno_actual/barrenos_menos1)"
      global internos= interpolate_pose (Linea12_A_p, Linea12_B_p, barreno_actual/barrenos_menos1)
      $ 1562 "internos" "breakAfter"
      movel(internos, a=0.5, v=0.1)
      $ 1563 "'desbaste_inicial'"
      # 'desbaste_inicial'
      $ 1564 "bajada_broca≔p[0,0,-0.024,0,0,0]"
      global bajada_broca=p[0,0,-0.024,0,0,0]
      $ 1565 "bajada≔p[0,0,0.024,0,0,0]"
      global bajada=p[0,0,0.024,0,0,0]
      $ 1566 "Direction: Base Z-"
      global move_thread_flag_1566=0
      thread move_thread_1566():
        enter_critical
        move_thread_flag_1566 = 1
        local towardsPos=calculate_point_to_move_towards(p[0.0,0.0,0.0,0.0,0.0,0.0], [0.0,0.0,-1.0], 0.071)
        movel(towardsPos, a=0.15, v=0.1)
        move_thread_flag_1566 = 2
        exit_critical
      end
      move_thread_flag_1566 = 0
      move_thread_han_1566 = run move_thread_1566()
      while (True):
        sleep(1.0E-10)
        if (move_thread_flag_1566 > 1):
          join move_thread_han_1566
          $ 1567 "Until (distance)"
          break
        end
        sync()
      end
      $ 1568 "Direction: Base Z-"
      global move_thread_flag_1568=0
      thread move_thread_1568():
        enter_critical
        move_thread_flag_1568 = 1
        local towardsPos=calculate_point_to_move_towards(p[0.0,0.0,0.0,0.0,0.0,0.0], [0.0,0.0,-1.0], 1000.0)
        movel(towardsPos, a=0.007, v=0.007)
        move_thread_flag_1568 = 2
        exit_critical
      end
      move_thread_flag_1568 = 0
      move_thread_han_1568 = run move_thread_1568()
      while (True):
        local targetTcpDirection=get_target_tcp_speed()
        local stepsToRetract=tool_contact(direction=targetTcpDirection)
        if (stepsToRetract > 0):
          kill move_thread_han_1568
          stopl(0.02)
          local backTrackMovement=get_actual_joint_positions_history(stepsToRetract)
          local contactPose=get_forward_kin(backTrackMovement)
          local posDir=[targetTcpDirection[0],targetTcpDirection[1],targetTcpDirection[2]]
          local retractTo=contactPose
          if (norm(posDir) > 1e-6):
            local normalizedPosDir=normalize(posDir)
            local additionalRetraction=p[normalizedPosDir[0] * 0.0, normalizedPosDir[1] * 0.0, normalizedPosDir[2] * 0.0, 0, 0, 0]
            retractTo = pose_sub(contactPose, additionalRetraction)
          end
          movel(retractTo, a=0.02, v=0.1)
          $ 1569 "Until (tool_contact_detection)"
          break
        end
        sync()
      end
      $ 1570 "Popup: punto contacto alanzdo"
      popup("punto contacto alanzdo", "Mensaje", False, False, blocking=True)
      $ 1571 "Direction: Base Z+"
      global move_thread_flag_1571=0
      thread move_thread_1571():
        enter_critical
        move_thread_flag_1571 = 1
        local towardsPos=calculate_point_to_move_towards(p[0.0,0.0,0.0,0.0,0.0,0.0], [0.0,0.0,1.0], 0.002)
        movel(towardsPos, a=0.005, v=0.003)
        move_thread_flag_1571 = 2
        exit_critical
      end
      move_thread_flag_1571 = 0
      move_thread_han_1571 = run move_thread_1571()
      while (True):
        sleep(1.0E-10)
        if (move_thread_flag_1571 > 1):
          join move_thread_han_1571
          $ 1572 "Until (distance)"
          break
        end
        sync()
      end
      $ 1573 "Wait: 0.3"
      sleep(0.3)
      $ 1574 "Set CO[1]=Encender"
      set_configurable_digital_out(1, True)
      $ 1575 "Wait: 0.3"
      sleep(0.3)
      $ 1576 "Loop 1 times"
      Loop_126 = 0
      while (Loop_126 < 1):
        $ 1577 "bajar≔pose_add(get_actual_tcp_pose(), bajada_broca)"
        global bajar= pose_add ( get_actual_tcp_pose (), bajada_broca)
        $ 1578 "bajar" "breakAfter"
        movel(bajar, a=0.004, v=0.004)
        $ 1579 "subir≔pose_sub(get_actual_tcp_pose(), bajada_broca)"
        global subir= pose_sub ( get_actual_tcp_pose (), bajada_broca)
        $ 1580 "Direction: Base Z+"
        global move_thread_flag_1580=0
        thread move_thread_1580():
          enter_critical
          move_thread_flag_1580 = 1
          local towardsPos=calculate_point_to_move_towards(p[0.0,0.0,0.0,0.0,0.0,0.0], [0.0,0.0,1.0], 0.002)
          movel(towardsPos, a=0.015, v=0.015)
          move_thread_flag_1580 = 2
          exit_critical
        end
        move_thread_flag_1580 = 0
        move_thread_han_1580 = run move_thread_1580()
        while (True):
          sleep(1.0E-10)
          if (move_thread_flag_1580 > 1):
            join move_thread_han_1580
            $ 1581 "Until (distance)"
            break
          end
          sync()
        end
        $ 1582 "Set CO[1]=Apagar"
        set_configurable_digital_out(1, False)
        $ 1583 "subir" "breakAfter"
        movel(subir, a=0.015, v=0.015)
        $ 1584 "bajada_broca≔pose_sub(bajada_broca, bajada)"
        global bajada_broca= pose_sub (bajada_broca, bajada)
        Loop_126 = Loop_126 + 1
      end
      $ 1585 "Direction: Base Z+"
      global move_thread_flag_1585=0
      thread move_thread_1585():
        enter_critical
        move_thread_flag_1585 = 1
        local towardsPos=calculate_point_to_move_towards(p[0.0,0.0,0.0,0.0,0.0,0.0], [0.0,0.0,1.0], 0.08)
        movel(towardsPos, a=0.15, v=0.1)
        move_thread_flag_1585 = 2
        exit_critical
      end
      move_thread_flag_1585 = 0
      move_thread_han_1585 = run move_thread_1585()
      while (True):
        sleep(1.0E-10)
        if (move_thread_flag_1585 > 1):
          join move_thread_han_1585
          $ 1586 "Until (distance)"
          break
        end
        sync()
      end
      $ 1587 "Set CO[1]=Apagar"
      set_configurable_digital_out(1, False)
      $ 1588 "barreno_actual≔barreno_actual+1"
      global barreno_actual=barreno_actual+1
    end
    $ 1591 "Popup: Linea12 con chica Terminada!"
    popup("Linea12 con chica Terminada!", "Mensaje", False, False, blocking=True)
    $ 1592 "Linea13"
    $ 1593 "Marcar_puntos"
    $ 1594 "MoveL"
    $ 1595 "Linea13_A" "breakAfter"
    movel(Linea13_A_p, a=0.5, v=0.1)
    $ 1596 "bajada_comprobacion"
    $ 1597 "Direction: Base Z-"
    global move_thread_flag_1597=0
    thread move_thread_1597():
      enter_critical
      move_thread_flag_1597 = 1
      local towardsPos=calculate_point_to_move_towards(p[0.0,0.0,0.0,0.0,0.0,0.0], [0.0,0.0,-1.0], 0.071)
      movel(towardsPos, a=0.15, v=0.1)
      move_thread_flag_1597 = 2
      exit_critical
    end
    move_thread_flag_1597 = 0
    move_thread_han_1597 = run move_thread_1597()
    while (True):
      sleep(1.0E-10)
      if (move_thread_flag_1597 > 1):
        join move_thread_han_1597
        $ 1598 "Until (distance)"
        break
      end
      sync()
    end
    $ 1599 "Direction: Base Z-"
    global move_thread_flag_1599=0
    thread move_thread_1599():
      enter_critical
      move_thread_flag_1599 = 1
      local towardsPos=calculate_point_to_move_towards(p[0.0,0.0,0.0,0.0,0.0,0.0], [0.0,0.0,-1.0], 1000.0)
      movel(towardsPos, a=0.007, v=0.007)
      move_thread_flag_1599 = 2
      exit_critical
    end
    move_thread_flag_1599 = 0
    move_thread_han_1599 = run move_thread_1599()
    while (True):
      local targetTcpDirection=get_target_tcp_speed()
      local stepsToRetract=tool_contact(direction=targetTcpDirection)
      if (stepsToRetract > 0):
        kill move_thread_han_1599
        stopl(0.02)
        local backTrackMovement=get_actual_joint_positions_history(stepsToRetract)
        local contactPose=get_forward_kin(backTrackMovement)
        local posDir=[targetTcpDirection[0],targetTcpDirection[1],targetTcpDirection[2]]
        local retractTo=contactPose
        if (norm(posDir) > 1e-6):
          local normalizedPosDir=normalize(posDir)
          local additionalRetraction=p[normalizedPosDir[0] * 0.0, normalizedPosDir[1] * 0.0, normalizedPosDir[2] * 0.0, 0, 0, 0]
          retractTo = pose_sub(contactPose, additionalRetraction)
        end
        movel(retractTo, a=0.02, v=0.1)
        $ 1600 "Until (tool_contact_detection)"
        break
      end
      sync()
    end
    $ 1601 "Direction: Base Z+"
    global move_thread_flag_1601=0
    thread move_thread_1601():
      enter_critical
      move_thread_flag_1601 = 1
      local towardsPos=calculate_point_to_move_towards(p[0.0,0.0,0.0,0.0,0.0,0.0], [0.0,0.0,1.0], 0.08)
      movel(towardsPos, a=0.15, v=0.1)
      move_thread_flag_1601 = 2
      exit_critical
    end
    move_thread_flag_1601 = 0
    move_thread_han_1601 = run move_thread_1601()
    while (True):
      sleep(1.0E-10)
      if (move_thread_flag_1601 > 1):
        join move_thread_han_1601
        $ 1602 "Until (distance)"
        break
      end
      sync()
    end
    $ 1603 "Linea13_B" "breakAfter"
    movel(Linea13_B_p, a=0.5, v=0.1)
    $ 1604 "bajada_comprobacion"
    $ 1605 "Direction: Base Z-"
    global move_thread_flag_1605=0
    thread move_thread_1605():
      enter_critical
      move_thread_flag_1605 = 1
      local towardsPos=calculate_point_to_move_towards(p[0.0,0.0,0.0,0.0,0.0,0.0], [0.0,0.0,-1.0], 0.071)
      movel(towardsPos, a=0.15, v=0.1)
      move_thread_flag_1605 = 2
      exit_critical
    end
    move_thread_flag_1605 = 0
    move_thread_han_1605 = run move_thread_1605()
    while (True):
      sleep(1.0E-10)
      if (move_thread_flag_1605 > 1):
        join move_thread_han_1605
        $ 1606 "Until (distance)"
        break
      end
      sync()
    end
    $ 1607 "Direction: Base Z-"
    global move_thread_flag_1607=0
    thread move_thread_1607():
      enter_critical
      move_thread_flag_1607 = 1
      local towardsPos=calculate_point_to_move_towards(p[0.0,0.0,0.0,0.0,0.0,0.0], [0.0,0.0,-1.0], 1000.0)
      movel(towardsPos, a=0.007, v=0.007)
      move_thread_flag_1607 = 2
      exit_critical
    end
    move_thread_flag_1607 = 0
    move_thread_han_1607 = run move_thread_1607()
    while (True):
      local targetTcpDirection=get_target_tcp_speed()
      local stepsToRetract=tool_contact(direction=targetTcpDirection)
      if (stepsToRetract > 0):
        kill move_thread_han_1607
        stopl(0.02)
        local backTrackMovement=get_actual_joint_positions_history(stepsToRetract)
        local contactPose=get_forward_kin(backTrackMovement)
        local posDir=[targetTcpDirection[0],targetTcpDirection[1],targetTcpDirection[2]]
        local retractTo=contactPose
        if (norm(posDir) > 1e-6):
          local normalizedPosDir=normalize(posDir)
          local additionalRetraction=p[normalizedPosDir[0] * 0.0, normalizedPosDir[1] * 0.0, normalizedPosDir[2] * 0.0, 0, 0, 0]
          retractTo = pose_sub(contactPose, additionalRetraction)
        end
        movel(retractTo, a=0.02, v=0.1)
        $ 1608 "Until (tool_contact_detection)"
        break
      end
      sync()
    end
    $ 1609 "Direction: Base Z+"
    global move_thread_flag_1609=0
    thread move_thread_1609():
      enter_critical
      move_thread_flag_1609 = 1
      local towardsPos=calculate_point_to_move_towards(p[0.0,0.0,0.0,0.0,0.0,0.0], [0.0,0.0,1.0], 0.08)
      movel(towardsPos, a=0.15, v=0.1)
      move_thread_flag_1609 = 2
      exit_critical
    end
    move_thread_flag_1609 = 0
    move_thread_han_1609 = run move_thread_1609()
    while (True):
      sleep(1.0E-10)
      if (move_thread_flag_1609 > 1):
        join move_thread_han_1609
        $ 1610 "Until (distance)"
        break
      end
      sync()
    end
    $ 1611 "AB"
    $ 1612 "'desbaste_inicial'"
    # 'desbaste_inicial'
    $ 1613 "bajada_broca≔p[0,0,-0.008,0,0,0]"
    global bajada_broca=p[0,0,-0.008,0,0,0]
    $ 1614 "barrenos_menos1≔2"
    global barrenos_menos1=2
    $ 1615 "barreno_actual≔0"
    global barreno_actual=0
    $ 1616 "Loop barreno_actual≤barrenos_menos1"
    while (barreno_actual <= barrenos_menos1):
      $ 1617 "Perforacion"
      $ 1618 "MoveL"
      $ 1621 "internos≔interpolate_pose(Linea13_A, Linea13_B, barreno_actual/barrenos_menos1)"
      global internos= interpolate_pose (Linea13_A_p, Linea13_B_p, barreno_actual/barrenos_menos1)
      $ 1622 "internos" "breakAfter"
      movel(internos, a=0.5, v=0.1)
      $ 1623 "'desbaste_inicial'"
      # 'desbaste_inicial'
      $ 1624 "bajada_broca≔p[0,0,-0.024,0,0,0]"
      global bajada_broca=p[0,0,-0.024,0,0,0]
      $ 1625 "bajada≔p[0,0,0.024,0,0,0]"
      global bajada=p[0,0,0.024,0,0,0]
      $ 1626 "Direction: Base Z-"
      global move_thread_flag_1626=0
      thread move_thread_1626():
        enter_critical
        move_thread_flag_1626 = 1
        local towardsPos=calculate_point_to_move_towards(p[0.0,0.0,0.0,0.0,0.0,0.0], [0.0,0.0,-1.0], 0.071)
        movel(towardsPos, a=0.15, v=0.1)
        move_thread_flag_1626 = 2
        exit_critical
      end
      move_thread_flag_1626 = 0
      move_thread_han_1626 = run move_thread_1626()
      while (True):
        sleep(1.0E-10)
        if (move_thread_flag_1626 > 1):
          join move_thread_han_1626
          $ 1627 "Until (distance)"
          break
